ACTION An_Conditions:
//正极纠偏平台允许放料条件
IF  NOT Mach_Control.An_b.An_deviationFalg AND arrAxisCtrl[AxiseNo.AxisName.AndeviationX1].Status.Homed AND NOT arrAxisCtrl[AxiseNo.AxisName.AndeviationX1].Status.Error AND 
	arrAxisCtrl[AxiseNo.AxisName.AndeviationX1].Status.NoMoving AND arrAxisCtrl[AxiseNo.AxisName.AndeviationX1].Cmd.arrbRealPoint[1] AND 
	arrAxisCtrl[AxiseNo.AxisName.AndeviationX2].Status.Homed AND NOT arrAxisCtrl[AxiseNo.AxisName.AndeviationX2].Status.Error AND 
	arrAxisCtrl[AxiseNo.AxisName.AndeviationX2].Status.NoMoving AND arrAxisCtrl[AxiseNo.AxisName.AndeviationX2].Cmd.arrbRealPoint[1] AND 
	arrAxisCtrl[AxiseNo.AxisName.AndeviationY].Status.Homed AND NOT arrAxisCtrl[AxiseNo.AxisName.AndeviationY].Status.Error AND 
	arrAxisCtrl[AxiseNo.AxisName.AndeviationY].Status.NoMoving AND arrAxisCtrl[AxiseNo.AxisName.AndeviationY].Cmd.arrbRealPoint[1] THEN
	Mach_Control.An_b.An_deviationFPOK:=TRUE;
ELSE
	Mach_Control.An_b.An_deviationFPOK:=FALSE;
END_IF 
(*
//正极纠偏平台允许取料条件
IF Mach_Control.An_b.An_deviationFalg AND  (Mach_Control.An_b.An_deviationDone OR Mach_Control.U.CCD_ChosesHMI OR Mach_Control.U.EmptyRunMode) THEN
	Mach_Control.An_b.An_deviationDPOK:=TRUE;
ELSE
	Mach_Control.An_b.An_deviationDPOK:=FALSE;
END_IF
*)
//正极送片搬运平移在安全位，正极送片升降在安全位，允许正极叠片搬运平移到纠偏位
IF arrAxisCtrl[AxiseNo.AxisName.AnCarryingLine].Status.Homed AND arrAxisCtrl[AxiseNo.AxisName.AnCarryingLine].Status.NoMoving AND arrAxisCtrl[AxiseNo.AxisName.AnCarryingLine].Cmd.arrbRealPoint[1] AND 
 	arrAxisCtrl[AxiseNo.AxisName.AnDTCarryingUpDown].Status.Homed AND arrAxisCtrl[AxiseNo.AxisName.AnDTCarryingUpDown].Status.NoMoving AND arrAxisCtrl[AxiseNo.AxisName.AnDTCarryingUpDown].Cmd.arrbRealPoint[1] THEN
	Mach_Control.An_b.CarryingSafepos[0]:=TRUE;
ELSE
	Mach_Control.An_b.CarryingSafepos[0]:=FALSE;
END_IF
//正极隔膜平移在负极片位、正极送片搬运升降在安全位，允许正极叠片搬动至叠台位
IF arrAxisCtrl[AxiseNo.AxisName.SEPTATLine].Status.Homed AND arrAxisCtrl[AxiseNo.AxisName.SEPTATLine].Status.NoMoving AND arrAxisCtrl[AxiseNo.AxisName.SEPTATLine].Cmd.arrbRealPoint[2] AND 
	 	arrAxisCtrl[AxiseNo.AxisName.AnDTCarryingUpDown].Status.Homed AND arrAxisCtrl[AxiseNo.AxisName.AnDTCarryingUpDown].Status.NoMoving AND arrAxisCtrl[AxiseNo.AxisName.AnDTCarryingUpDown].Cmd.arrbRealPoint[1] THEN
	Mach_Control.An_b.CarryingSafepos[1]:=TRUE;
ELSE		
	Mach_Control.An_b.CarryingSafepos[1]:=FALSE;
END_IF
//正极送片搬运升降在安全位，允许正极送片搬运平移至取流水线极片位
IF  arrAxisCtrl[AxiseNo.AxisName.AnCarryingUpDown].Status.Homed AND arrAxisCtrl[AxiseNo.AxisName.AnCarryingUpDown].Status.NoMoving AND arrAxisCtrl[AxiseNo.AxisName.AnCarryingUpDown].Cmd.arrbRealPoint[1] THEN
		Mach_Control.An_b.CarryingSafepos[2]:=TRUE;
ELSE
		Mach_Control.An_b.CarryingSafepos[2]:=FALSE;	
END_IF
//正极送片搬运升降在安全位、正极叠片搬运平移在安全位，允许正极送片搬运平移纠偏位
IF  arrAxisCtrl[AxiseNo.AxisName.AnCarryingUpDown].Status.Homed AND arrAxisCtrl[AxiseNo.AxisName.AnCarryingUpDown].Status.NoMoving AND arrAxisCtrl[AxiseNo.AxisName.AnCarryingUpDown].Cmd.arrbRealPoint[1] AND 
 	arrAxisCtrl[AxiseNo.AxisName.AnDTCarryingLine].Status.Homed AND arrAxisCtrl[AxiseNo.AxisName.AnDTCarryingLine].Status.NoMoving AND arrAxisCtrl[AxiseNo.AxisName.AnDTCarryingLine].Cmd.arrbRealPoint[2]  THEN
		Mach_Control.An_b.CarryingSafepos[3]:=TRUE;
ELSE
		Mach_Control.An_b.CarryingSafepos[3]:=FALSE;	
END_IF
//允许正极纠偏平台移动
IF arrAxisCtrl[AxiseNo.AxisName.AnCarryingUpDown].Status.Homed AND arrAxisCtrl[AxiseNo.AxisName.AnCarryingLine].Status.Homed AND 
	((arrAxisCtrl[AxiseNo.AxisName.AnCarryingUpDown].Status.fSetPos<=arrAxisPar[AxiseNo.AxisName.AnCarryingUpDown].arrTargetPoint[4]+2) OR arrAxisCtrl[AxiseNo.AxisName.AnCarryingLine].Cmd.arrbGoSetPos[1]) AND 
	((arrAxisCtrl[AxiseNo.AxisName.AnDTCarryingUpDown].Status.fSetPos<=arrAxisPar[AxiseNo.AxisName.AnDTCarryingUpDown].arrTargetPoint[4]+2) OR arrAxisCtrl[AxiseNo.AxisName.AnDTCarryingLine].Cmd.arrbGoSetPos[2])THEN
	Mach_Control.An_b.CarryingSafepos[4]:=TRUE;
ELSE
	Mach_Control.An_b.CarryingSafepos[4]:=FALSE;
END_IF
//正极取流水线机械手在安全位，允许模切流水线移动
(*
IF arrAxisCtrl[AxiseNo.AxisName.AnCarryingUpDown].Status.Homed AND NOT Mach_Control.An_b.An_MainBelting AND
	(arrAxisCtrl[AxiseNo.AxisName.AnCarryingUpDown].Status.fSetPos<=arrAxisPar[AxiseNo.AxisName.AnCarryingUpDown].arrTargetPoint[4]+0.2 OR arrAxisCtrl[AxiseNo.AxisName.AnCarryingLine].Cmd.arrbRealPoint[2]) THEN
	Mach_Control.An_b.AN_BeltSafe:=TRUE;
ELSE
	Mach_Control.An_b.AN_BeltSafe:=FALSE;
END_IF
*)
(*
IF  Mach_Control.An_b.An_MainBelting  THEN
	Mach_Control.An_b.AN_BeltSafe:=TRUE;
ELSIF NOT Mach_Control.An_b.An_MainBelting AND  arrAxisCtrl[AxiseNo.AxisName.AnCarryingUpDown].Cmd.arrbRealPoint[4] THEN
	Mach_Control.An_b.AN_BeltSafe:=FALSE;
END_IF
*)
IF  Mach_Control.An_b.An_MainBelting  THEN
	Mach_Control.An_b.AN_BeltSafe:=TRUE;
ELSE
	Mach_Control.An_b.AN_BeltSafe:=FALSE;
END_IF

//正极主流水线取片完成延时复位
An_BeltTon(IN:=Mach_Control.An_b.AN_BeltDone , PT:=T#0.1S , Q=> , ET=> );
IF An_BeltTon.Q THEN
	Mach_Control.An_b.AN_BeltDone :=FALSE;
END_IF


//正极跳取条件1:空跑(空叠隔膜)
An_JumpRules[1]:=Mach_Control.U.EmptyRunMode OR (Mach_Control.DT_b.SinStepMode AND An_Step0<>150);
//正极跳取条件2:手动
An_JumpRules[2]:=Mach_Control.U.DT_iMode<>1;
//正极跳取条件3:叠完电芯后空叠隔膜
An_JumpRules[3]:=Mach_Control.DT_b.DP_Mode AND Mach_Control.An_b.An_Quantited=Par.stDT_date.An_Quantity AND Par.stDT_date.An_Quantity<>0  ;
//正极跳取条件4:叠完电芯后下料
An_JumpRules[4]:=DP_Step0>=6000;//(DP_Step0>=6030 AND DP_Step0<6041) ;
//正极跳取条件5:正极剔废,
An_JumpRules[5]:=(An_Step2<>0 AND An_Step2<>6666) ; 
//正极跳取条件6:接带、蓝胶判断
An_JumpRules[6]:=Bnt_Blueflaging AND Mach_Control.Ca_b.Ca_Quantited>=Par.stDT_date.DT_Overhang_SUM AND Par.stDT_date.DT_Overhang_SUM>0 
				AND Mach_Control.Ca_b.Ca_Quantited>Mach_Control.An_b.An_Quantited AND An_StandbyStep1<1000;//已经进入取片流程则取完当前片
//正极跳取条件7:取片升降有片
An_JumpRules[7]:= Mach_Control.An_b.An_CarryingFalg  ;
//正极跳取条件8:对齐度踢废
An_JumpRules[8]:=Mach_Control.DT_b.DT_Oerhang_Z=2 AND  Par.stDT_date.DT_Overhang_SUM>0 AND Mach_Control.Ca_b.Ca_Quantited>=Par.stDT_date.DT_Overhang_SUM
				AND Mach_Control.An_b.An_Quantited<Mach_Control.Ca_b.Ca_Quantited  AND  Mach_Control.DT_b.DT_CellNG_TF AND Mach_Control.DT_b.Overhang_TF 
				AND((NOT Mach_Control.DT_b.FirstEmpFold AND   bFirstFoldFinish[1]) OR (Mach_Control.DT_b.FirstEmpFold)) AND An_StandbyStep1<1000;//已经进入取片流程则取完当前片
//正极跳取条件9:负极剔废
An_JumpRules[9]:=(Ca_Step2<>0 AND Ca_Step2<>6666) ;
//正极跳取条件10:首层空叠隔膜流程
An_JumpRules[10]:=NOT bFirstFoldFinish[1]AND NOT Mach_Control.DT_b.FirstEmpFold ; 			
//正极跳取条件
Mach_Control.An_b.JumpPiceReady:=An_JumpRules[1] OR An_JumpRules[2] OR An_JumpRules[3] OR An_JumpRules[4] OR An_JumpRules[5]
				OR An_JumpRules[6] OR An_JumpRules[7] OR An_JumpRules[8]  OR An_JumpRules[9] OR An_JumpRules[10] OR DP_Step0=162;	//速度不一样如果平移没到位放弃取片 20240509 CF	
//正极取片条件
Mach_Control.An_b.GetPiceReady:=NOT Mach_Control.An_b.JumpPiceReady (*AND  arrAxisCtrl[AxiseNo.AxisName.AnCarryingUpDown].Cmd.arrbRealPoint[4]*)
				AND ABS(arrAxisCtrl[AxiseNo.AxisName.AnCarryingLine].Status.fSetPos-arrAxisPar[AxiseNo.AxisName.AnCarryingLine].arrTargetPoint[1])<0.5 AND  arrAxisCtrl[AxiseNo.AxisName.AnCarryingWhirling].Cmd.arrbRealPoint[1]
				AND Mach_Control.U.DT_iMode=1 AND NOT Mach_Control.An_b.An_CarryingFalg ;//20240509 CF 升降位置判断屏蔽
		
(*				
////////////////判断叠台是否需要极片
//南昌原版
JumpPiceReady_temp1:=Mach_Control.An_b.An_Quantited<Mach_Control.Ca_b.Ca_Quantited AND Par.stDT_date.An_Quantity<>0  AND
 	 				 Par.stDT_date.Ca_Quantity <>0 AND  Mach_Control.DT_b.DT_CellNG_TF AND
	 				 Mach_Control.Ca_b.Ca_Quantited>=Par.stDT_date.DT_Overhang_SUM AND Par.stDT_date.DT_Overhang_SUM>0  AND
     				 Mach_Control.DT_b.DT_Oerhang_Z=2 AND  NOT Mach_Control.U.EmptyRunMode;

JumpPiceReady_temp2:=Bnt_Blueflaging AND ((Mach_Control.An_b.An_Quantited=0 AND Mach_Control.Ca_b.Ca_Quantited=0) OR
 					 Mach_Control.Ca_b.Ca_Quantited>Mach_Control.An_b.An_Quantited);

JumpPiceReady_temp3:= Mach_Control.An_b.An_Quantited >= Par.stDT_date.An_Quantity  AND
  					  Mach_Control.Ca_b.Ca_Quantited >= Par.stDT_date.Ca_Quantity AND
                      Par.stDT_date.An_Quantity<>0  AND Par.stDT_date.Ca_Quantity <>0;
					  
JumpPiceReady_temp4:= (Ca_Step2<>0 AND Ca_Step2<>6666 AND Mach_Control.U.DT_iMode=1)OR (Mach_Control.An_b.An_Quantited >= Par.stDT_date.An_Quantity 
					 AND  Mach_Control.Ca_b.Ca_Quantited >= (Par.stDT_date.Ca_Quantity-1)) OR
					   (Bnt_Blueflaging AND Mach_Control.Ca_b.Ca_Quantited>=Par.stDT_date.DT_Overhang_SUM AND Par.stDT_date.DT_Overhang_SUM>0);

					   
//正极送片搬运搬运取片准备好
IF Mach_Control.U.DT_iMode=1 AND NOT Mach_Control.An_b.An_CarryingFalg AND NOT JumpPiceReady_temp4 AND (DP_Step0<>6030 AND DP_Step0<>6040 AND 
Mach_Control.An_b.An_Quantited <= Par.stDT_date.An_Quantity  AND  Mach_Control.Ca_b.Ca_Quantited < Par.stDT_date.Ca_Quantity) AND
   arrAxisCtrl[AxiseNo.AxisName.AnCarryingUpDown].Cmd.arrbRealPoint[4] AND arrAxisCtrl[AxiseNo.AxisName.AnCarryingUpDown].Status.Homed AND
   arrAxisCtrl[AxiseNo.AxisName.AnCarryingLine].Cmd.arrbRealPoint[1] AND arrAxisCtrl[AxiseNo.AxisName.AnCarryingLine].Status.Homed AND
   arrAxisCtrl[AxiseNo.AxisName.AnCarryingWhirling].Cmd.arrbRealPoint[1]AND arrAxisCtrl[AxiseNo.AxisName.AnCarryingWhirling].Status.Homed  THEN
   Mach_Control.An_b.GetPiceReady:=TRUE;
ELSE
   Mach_Control.An_b.GetPiceReady:=FALSE;	
END_IF

//正极送片搬运不取片
IF Mach_Control.U.DT_iMode<>1 OR Mach_Control.An_b.An_CarryingFalg OR JumpPiceReady_temp1 OR JumpPiceReady_temp2 OR JumpPiceReady_temp3 OR JumpPiceReady_temp4 OR Mach_Control.U.EmptyRunMode THEN
	Mach_Control.An_b.JumpPiceReady:=TRUE;
ELSE
	Mach_Control.An_b.JumpPiceReady:=FALSE;	
END_IF


//合肥原版
(*
(********************正极取片准备好********************)															
Mach_Control.An_b.GetPiceReady:=NOT Mach_Control.An_b.JumpPiceReady AND 
							arrAxisCtrl[AxiseNo.AxisName.AnCarryingUpDown].Cmd.arrbRealPoint[4] AND arrAxisCtrl[AxiseNo.AxisName.AnCarryingUpDown].Status.Homed AND
							arrAxisCtrl[AxiseNo.AxisName.AnCarryingLine].Cmd.arrbRealPoint[1] AND arrAxisCtrl[AxiseNo.AxisName.AnCarryingLine].Status.Homed AND
							arrAxisCtrl[AxiseNo.AxisName.AnCarryingWhirling].Cmd.arrbRealPoint[1]AND arrAxisCtrl[AxiseNo.AxisName.AnCarryingWhirling].Status.Homed AND 
							(DP_Step0<>6030 AND DP_Step0<>6040)  ;													

(********************正极放弃取片********************)
Mach_Control.An_b.JumpPiceReady:=Mach_Control.U.DT_iMode<>1 OR Mach_Control.An_b.An_CarryingFalg OR Blueflaging OR Mach_Control.U.EmptyRunMode
															OR Mach_Control.An_b.An_Quantited=Par.stDT_date.An_Quantity;
*)

*)


/////////////////////////////////////////////////////////////
/////////////////////////////////////////////////////////
////////////////////////////////////////////电机条件
//正极送片搬运平移
IF arrAxisCtrl[AxiseNo.AxisName.AnCarryingUpDown].Status.fSetPos<=arrAxisPar[AxiseNo.AxisName.AnCarryingUpDown].arrTargetPoint[4]+1 AND
 	arrAxisCtrl[AxiseNo.AxisName.AnCarryingUpDown].Status.Homed AND arrAxisCtrl[AxiseNo.AxisName.AnCarryingUpDown].Status.NoMoving	AND Mach_Control.U.DT_iMode=3 THEN
arrAxisCtrl[AxiseNo.AxisName.AnCarryingLine].Cmd.Home_Condition:=TRUE;
ELSE
arrAxisCtrl[AxiseNo.AxisName.AnCarryingLine].Cmd.Home_Condition:=FALSE;	
END_IF

IF arrAxisCtrl[AxiseNo.AxisName.AnCarryingUpDown].Status.fSetPos<=arrAxisPar[AxiseNo.AxisName.AnCarryingUpDown].arrTargetPoint[4]+1 AND
	arrAxisCtrl[AxiseNo.AxisName.AnCarryingUpDown].Status.Homed AND arrAxisCtrl[AxiseNo.AxisName.AnCarryingUpDown].Status.NoMoving AND Mach_Control.U.DT_iMode=3 
    AND 	arrCyCtrl[arrCyNo.CylinderName.AnScrapbinCy].Io.DIOnSwitch  THEN
arrAxisCtrl[AxiseNo.AxisName.AnCarryingLine].Cmd.GoPoint_Condition[1]:=TRUE;
ELSE
arrAxisCtrl[AxiseNo.AxisName.AnCarryingLine].Cmd.GoPoint_Condition[1]:=FALSE;	
END_IF

IF arrAxisCtrl[AxiseNo.AxisName.AnCarryingUpDown].Status.fSetPos<=arrAxisPar[AxiseNo.AxisName.AnCarryingUpDown].arrTargetPoint[4]+1 AND arrAxisCtrl[AxiseNo.AxisName.AnCarryingUpDown].Status.Homed  AND
	 arrAxisCtrl[AxiseNo.AxisName.AnCarryingLine].Status.Homed AND Mach_Control.U.DT_iMode=3 AND 	arrCyCtrl[arrCyNo.CylinderName.AnScrapbinCy].Io.DIOnSwitch AND
	 arrAxisCtrl[AxiseNo.AxisName.AnDTCarryingLine].Status.Homed AND arrAxisCtrl[AxiseNo.AxisName.AnDTCarryingLine].Cmd.arrbRealPoint[2] THEN//比较值要根据实际值修改
	arrAxisCtrl[AxiseNo.AxisName.AnCarryingLine].Cmd.GoPoint_Condition[2]:=TRUE;
ELSE
	arrAxisCtrl[AxiseNo.AxisName.AnCarryingLine].Cmd.GoPoint_Condition[2]:=FALSE;	
END_IF

//正极送片搬运升降
IF Mach_Control.U.DT_iMode=3  THEN
	arrAxisCtrl[AxiseNo.AxisName.AnCarryingUpDown].Cmd.Home_Condition:=TRUE;
ELSE
	arrAxisCtrl[AxiseNo.AxisName.AnCarryingUpDown].Cmd.Home_Condition:=FALSE;	
END_IF

IF Mach_Control.U.DT_iMode=3 AND arrAxisCtrl[AxiseNo.AxisName.AnCarryingUpDown].Status.Homed THEN
	arrAxisCtrl[AxiseNo.AxisName.AnCarryingUpDown].Cmd.GoPoint_Condition[1]:=TRUE;
ELSE
	arrAxisCtrl[AxiseNo.AxisName.AnCarryingUpDown].Cmd.GoPoint_Condition[1]:=FALSE;	
END_IF

IF (*arrAxisCtrl[AxiseNo.AxisName.AnCarryingLine].Cmd.arrbRealPoint[1] AND*)  Mach_Control.U.DT_iMode=3 AND arrAxisCtrl[AxiseNo.AxisName.AnCarryingUpDown].Status.Homed THEN
	arrAxisCtrl[AxiseNo.AxisName.AnCarryingUpDown].Cmd.GoPoint_Condition[2]:=TRUE;
ELSE
	arrAxisCtrl[AxiseNo.AxisName.AnCarryingUpDown].Cmd.GoPoint_Condition[2]:=FALSE;	
END_IF

IF (*arrAxisCtrl[AxiseNo.AxisName.AnCarryingLine].Cmd.arrbRealPoint[2] AND*)  Mach_Control.U.DT_iMode=3 AND arrAxisCtrl[AxiseNo.AxisName.AnCarryingUpDown].Status.Homed THEN
	arrAxisCtrl[AxiseNo.AxisName.AnCarryingUpDown].Cmd.GoPoint_Condition[3]:=TRUE;
ELSE
	arrAxisCtrl[AxiseNo.AxisName.AnCarryingUpDown].Cmd.GoPoint_Condition[3]:=FALSE;	
END_IF

IF (*arrAxisCtrl[AxiseNo.AxisName.AnCarryingLine].Cmd.arrbRealPoint[1] AND*)  Mach_Control.U.DT_iMode=3 AND arrAxisCtrl[AxiseNo.AxisName.AnCarryingUpDown].Status.Homed THEN
	arrAxisCtrl[AxiseNo.AxisName.AnCarryingUpDown].Cmd.GoPoint_Condition[4]:=TRUE;
ELSE
	arrAxisCtrl[AxiseNo.AxisName.AnCarryingUpDown].Cmd.GoPoint_Condition[4]:=FALSE;	
END_IF

//正极送片搬运旋转
IF Mach_Control.U.DT_iMode=3 AND
 	arrAxisCtrl[AxiseNo.AxisName.AnCarryingUpDown].Status.fSetPos <= arrAxisPar[AxiseNo.AxisName.AnCarryingUpDown].arrTargetPoint[1]+1 AND 
	arrAxisCtrl[AxiseNo.AxisName.AnCarryingUpDown].Status.Homed AND arrCyCtrl[arrCyNo.CylinderName.AnScrapbinCy].Io.DIOnSwitch   THEN
	arrAxisCtrl[AxiseNo.AxisName.AnCarryingWhirling].Cmd.Home_Condition:=TRUE;
ELSE
	arrAxisCtrl[AxiseNo.AxisName.AnCarryingWhirling].Cmd.Home_Condition:=FALSE;	
END_IF


IF Mach_Control.U.DT_iMode=3 AND
 	arrAxisCtrl[AxiseNo.AxisName.AnCarryingUpDown].Status.fSetPos <= arrAxisPar[AxiseNo.AxisName.AnCarryingUpDown].arrTargetPoint[1]+1 AND 
	arrAxisCtrl[AxiseNo.AxisName.AnCarryingUpDown].Status.Homed AND arrCyCtrl[arrCyNo.CylinderName.AnScrapbinCy].Io.DIOnSwitch    THEN
	   arrAxisCtrl[AxiseNo.AxisName.AnCarryingWhirling].Cmd.JogP_Condition:=TRUE;
	   arrAxisCtrl[AxiseNo.AxisName.AnCarryingWhirling].Cmd.JogN_Condition:=TRUE;
 ELSE 
	   arrAxisCtrl[AxiseNo.AxisName.AnCarryingWhirling].Cmd.JogP_Condition:=FALSE;
	   arrAxisCtrl[AxiseNo.AxisName.AnCarryingWhirling].Cmd.JogN_Condition:=FALSE;
 END_IF

IF Mach_Control.U.DT_iMode=3 AND 
	(arrAxisCtrl[AxiseNo.AxisName.AnCarryingUpDown].Cmd.arrbRealPoint[1] (*OR arrAxisCtrl[AxiseNo.AxisName.AnCarryingUpDown].Cmd.arrbRealPoint[4]*))AND
	arrAxisCtrl[AxiseNo.AxisName.AnCarryingUpDown].Status.Homed AND arrAxisCtrl[AxiseNo.AxisName.AnCarryingWhirling].Status.Homed AND 
    arrCyCtrl[arrCyNo.CylinderName.AnScrapbinCy].Io.DIOnSwitch   THEN
	arrAxisCtrl[AxiseNo.AxisName.AnCarryingWhirling].Cmd.GoPoint_Condition[1]:=TRUE;
ELSE
	arrAxisCtrl[AxiseNo.AxisName.AnCarryingWhirling].Cmd.GoPoint_Condition[1]:=FALSE;	
END_IF

IF Mach_Control.U.DT_iMode=3 AND 
	(arrAxisCtrl[AxiseNo.AxisName.AnCarryingUpDown].Cmd.arrbRealPoint[1] (*OR arrAxisCtrl[AxiseNo.AxisName.AnCarryingUpDown].Cmd.arrbRealPoint[4]*)) AND
	arrAxisCtrl[AxiseNo.AxisName.AnCarryingUpDown].Status.Homed AND arrAxisCtrl[AxiseNo.AxisName.AnCarryingWhirling].Status.Homed AND
   arrCyCtrl[arrCyNo.CylinderName.AnScrapbinCy].Io.DIOnSwitch  THEN
	arrAxisCtrl[AxiseNo.AxisName.AnCarryingWhirling].Cmd.GoPoint_Condition[2]:=TRUE;
ELSE
	arrAxisCtrl[AxiseNo.AxisName.AnCarryingWhirling].Cmd.GoPoint_Condition[2]:=FALSE;	
END_IF

//正极纠偏平台X1
IF Mach_Control.U.DT_iMode=3  OR  (DP_Step0>=6015 AND   DP_Step0<=6041)   THEN
	arrAxisCtrl[AxiseNo.AxisName.AndeviationX1].Cmd.Home_Condition:=TRUE;
ELSE
	arrAxisCtrl[AxiseNo.AxisName.AndeviationX1].Cmd.Home_Condition:=FALSE;	
END_IF

IF Mach_Control.U.DT_iMode=3 AND arrAxisCtrl[AxiseNo.AxisName.AndeviationX1].Status.Homed THEN
	arrAxisCtrl[AxiseNo.AxisName.AndeviationX1].Cmd.GoPoint_Condition[1]:=TRUE;
ELSE
	arrAxisCtrl[AxiseNo.AxisName.AndeviationX1].Cmd.GoPoint_Condition[1]:=FALSE;	
END_IF

IF Mach_Control.U.DT_iMode=3 AND arrAxisCtrl[AxiseNo.AxisName.AndeviationX1].Status.Homed THEN
	arrAxisCtrl[AxiseNo.AxisName.AndeviationX1].Cmd.GoPoint_Condition[2]:=TRUE;
ELSE
	arrAxisCtrl[AxiseNo.AxisName.AndeviationX1].Cmd.GoPoint_Condition[2]:=FALSE;	
END_IF

IF Mach_Control.U.DT_iMode=3 AND arrAxisCtrl[AxiseNo.AxisName.AndeviationX1].Status.Homed THEN
	arrAxisCtrl[AxiseNo.AxisName.AndeviationX1].Cmd.GoPoint_Condition[3]:=TRUE;
ELSE
	arrAxisCtrl[AxiseNo.AxisName.AndeviationX1].Cmd.GoPoint_Condition[3]:=FALSE;	
END_IF

IF Mach_Control.U.DT_iMode=3 AND arrAxisCtrl[AxiseNo.AxisName.AndeviationX1].Status.Homed THEN
	arrAxisCtrl[AxiseNo.AxisName.AndeviationX1].Cmd.GoPoint_Condition[4]:=TRUE;
ELSE
	arrAxisCtrl[AxiseNo.AxisName.AndeviationX1].Cmd.GoPoint_Condition[4]:=FALSE;	
END_IF

IF Mach_Control.U.DT_iMode=3 AND arrAxisCtrl[AxiseNo.AxisName.AndeviationX1].Status.Homed THEN
	arrAxisCtrl[AxiseNo.AxisName.AndeviationX1].Cmd.GoPoint_Condition[5]:=TRUE;
ELSE
	arrAxisCtrl[AxiseNo.AxisName.AndeviationX1].Cmd.GoPoint_Condition[5]:=FALSE;	
END_IF

//正极纠偏平台X2
IF Mach_Control.U.DT_iMode=3  OR  (DP_Step0>=6015 AND   DP_Step0<=6041)   THEN
	arrAxisCtrl[AxiseNo.AxisName.AndeviationX2].Cmd.Home_Condition:=TRUE;
ELSE
	arrAxisCtrl[AxiseNo.AxisName.AndeviationX2].Cmd.Home_Condition:=FALSE;	
END_IF

IF Mach_Control.U.DT_iMode=3 AND arrAxisCtrl[AxiseNo.AxisName.AndeviationX2].Status.Homed THEN
	arrAxisCtrl[AxiseNo.AxisName.AndeviationX2].Cmd.GoPoint_Condition[1]:=TRUE;
ELSE
	arrAxisCtrl[AxiseNo.AxisName.AndeviationX2].Cmd.GoPoint_Condition[1]:=FALSE;	
END_IF

IF Mach_Control.U.DT_iMode=3 AND arrAxisCtrl[AxiseNo.AxisName.AndeviationX2].Status.Homed THEN
	arrAxisCtrl[AxiseNo.AxisName.AndeviationX2].Cmd.GoPoint_Condition[2]:=TRUE;
ELSE
	arrAxisCtrl[AxiseNo.AxisName.AndeviationX2].Cmd.GoPoint_Condition[2]:=FALSE;	
END_IF

IF Mach_Control.U.DT_iMode=3 AND arrAxisCtrl[AxiseNo.AxisName.AndeviationX2].Status.Homed THEN
	arrAxisCtrl[AxiseNo.AxisName.AndeviationX2].Cmd.GoPoint_Condition[3]:=TRUE;
ELSE
	arrAxisCtrl[AxiseNo.AxisName.AndeviationX2].Cmd.GoPoint_Condition[3]:=FALSE;	
END_IF

IF Mach_Control.U.DT_iMode=3 AND arrAxisCtrl[AxiseNo.AxisName.AndeviationX2].Status.Homed THEN
	arrAxisCtrl[AxiseNo.AxisName.AndeviationX2].Cmd.GoPoint_Condition[4]:=TRUE;
ELSE
	arrAxisCtrl[AxiseNo.AxisName.AndeviationX2].Cmd.GoPoint_Condition[4]:=FALSE;	
END_IF

IF Mach_Control.U.DT_iMode=3 AND arrAxisCtrl[AxiseNo.AxisName.AndeviationX2].Status.Homed THEN
	arrAxisCtrl[AxiseNo.AxisName.AndeviationX2].Cmd.GoPoint_Condition[5]:=TRUE;
ELSE
	arrAxisCtrl[AxiseNo.AxisName.AndeviationX2].Cmd.GoPoint_Condition[5]:=FALSE;	
END_IF

//正极纠偏平台Y
IF Mach_Control.U.DT_iMode=3  OR  (DP_Step0>=6015 AND   DP_Step0<=6041)   THEN
	arrAxisCtrl[AxiseNo.AxisName.AndeviationY].Cmd.Home_Condition:=TRUE;
ELSE
	arrAxisCtrl[AxiseNo.AxisName.AndeviationY].Cmd.Home_Condition:=FALSE;	
END_IF

IF Mach_Control.U.DT_iMode=3 AND arrAxisCtrl[AxiseNo.AxisName.AndeviationY].Status.Homed THEN
	arrAxisCtrl[AxiseNo.AxisName.AndeviationY].Cmd.GoPoint_Condition[1]:=TRUE;
ELSE
	arrAxisCtrl[AxiseNo.AxisName.AndeviationY].Cmd.GoPoint_Condition[1]:=FALSE;	
END_IF

IF Mach_Control.U.DT_iMode=3 AND arrAxisCtrl[AxiseNo.AxisName.AndeviationY].Status.Homed THEN
	arrAxisCtrl[AxiseNo.AxisName.AndeviationY].Cmd.GoPoint_Condition[2]:=TRUE;
ELSE
	arrAxisCtrl[AxiseNo.AxisName.AndeviationY].Cmd.GoPoint_Condition[2]:=FALSE;	
END_IF

IF Mach_Control.U.DT_iMode=3 AND arrAxisCtrl[AxiseNo.AxisName.AndeviationY].Status.Homed THEN
	arrAxisCtrl[AxiseNo.AxisName.AndeviationY].Cmd.GoPoint_Condition[3]:=TRUE;
ELSE
	arrAxisCtrl[AxiseNo.AxisName.AndeviationY].Cmd.GoPoint_Condition[3]:=FALSE;	
END_IF

IF Mach_Control.U.DT_iMode=3 AND arrAxisCtrl[AxiseNo.AxisName.AndeviationY].Status.Homed THEN
	arrAxisCtrl[AxiseNo.AxisName.AndeviationY].Cmd.GoPoint_Condition[4]:=TRUE;
ELSE
	arrAxisCtrl[AxiseNo.AxisName.AndeviationY].Cmd.GoPoint_Condition[4]:=FALSE;	
END_IF

IF Mach_Control.U.DT_iMode=3 AND arrAxisCtrl[AxiseNo.AxisName.AndeviationY].Status.Homed THEN
	arrAxisCtrl[AxiseNo.AxisName.AndeviationY].Cmd.GoPoint_Condition[5]:=TRUE;
ELSE
	arrAxisCtrl[AxiseNo.AxisName.AndeviationY].Cmd.GoPoint_Condition[5]:=FALSE;	
END_IF

//正极叠台搬运平移1
IF Mach_Control.U.DT_iMode=3 AND arrAxisCtrl[AxiseNo.AxisName.AnDTCarryingUpDown].Status.Homed AND
	arrAxisCtrl[AxiseNo.AxisName.AnDTCarryingUpDown].Status.fSetPos<= arrAxisPar[AxiseNo.AxisName.AnDTCarryingUpDown].arrTargetPoint[4]+1 AND
	arrAxisCtrl[AxiseNo.AxisName.AnCarryingLine].Status.fSetPos<=arrAxisPar[AxiseNo.AxisName.AnCarryingLine].arrTargetPoint[1] AND 
	arrCyCtrl[arrCyNo.CylinderName.AnScrapbinCy].Io.DIOnSwitch  AND NOT arrCyCtrl[arrCyNo.CylinderName.AnScrapbinCy].Io.DIOFFSwitch AND
	arrAxisCtrl[AxiseNo.AxisName.AnCarryingLine].Status.Homed AND arrAxisCtrl[AxiseNo.AxisName.AnCarryingLine].Status.NoMoving THEN
	arrAxisCtrl[AxiseNo.AxisName.AnDTCarryingLine].Cmd.Home_Condition:=TRUE;
ELSE
	arrAxisCtrl[AxiseNo.AxisName.AnDTCarryingLine].Cmd.Home_Condition:=FALSE;	
END_IF

IF Mach_Control.U.DT_iMode=3 AND arrCyCtrl[arrCyNo.CylinderName.AnScrapbinCy].Status.ONState THEN
   arrAxisCtrl[AxiseNo.AxisName.AnDTCarryingLine].Cmd.JogP_Condition:=TRUE;
   arrAxisCtrl[AxiseNo.AxisName.AnDTCarryingLine].Cmd.JogN_Condition:=TRUE;
   ELSE 
   arrAxisCtrl[AxiseNo.AxisName.AnDTCarryingLine].Cmd.JogP_Condition:=FALSE;
   arrAxisCtrl[AxiseNo.AxisName.AnDTCarryingLine].Cmd.JogN_Condition:=FALSE;
 END_IF

IF Mach_Control.U.DT_iMode=3 AND arrAxisCtrl[AxiseNo.AxisName.AnDTCarryingUpDown].Status.Homed AND
	arrAxisCtrl[AxiseNo.AxisName.AnDTCarryingUpDown].Status.fSetPos<= arrAxisPar[AxiseNo.AxisName.AnDTCarryingUpDown].arrTargetPoint[4]+1 AND
	arrAxisCtrl[AxiseNo.AxisName.AnCarryingLine].Cmd.arrbRealPoint[1] AND arrCyCtrl[arrCyNo.CylinderName.AnScrapbinCy].Status.ONState  THEN
	arrAxisCtrl[AxiseNo.AxisName.AnDTCarryingLine].Cmd.GoPoint_Condition[1]:=TRUE;
ELSE
	arrAxisCtrl[AxiseNo.AxisName.AnDTCarryingLine].Cmd.GoPoint_Condition[1]:=FALSE;	
END_IF

IF Mach_Control.U.DT_iMode=3 AND arrAxisCtrl[AxiseNo.AxisName.AnDTCarryingUpDown].Status.Homed AND
	arrAxisCtrl[AxiseNo.AxisName.AnDTCarryingUpDown].Status.fSetPos<= arrAxisPar[AxiseNo.AxisName.AnDTCarryingUpDown].arrTargetPoint[4]+1 AND
 	arrAxisCtrl[AxiseNo.AxisName.AnDTCarryingLine].Status.Homed AND arrAxisCtrl[AxiseNo.AxisName.SEPTATLine].Cmd.arrbRealPoint[2] AND
    arrCyCtrl[arrCyNo.CylinderName.AnScrapbinCy].Status.ONState THEN
	arrAxisCtrl[AxiseNo.AxisName.AnDTCarryingLine].Cmd.GoPoint_Condition[2]:=TRUE;
ELSE
	arrAxisCtrl[AxiseNo.AxisName.AnDTCarryingLine].Cmd.GoPoint_Condition[2]:=FALSE;	
END_IF


//正极叠台搬运升降1
IF Mach_Control.U.DT_iMode=3  THEN
	arrAxisCtrl[AxiseNo.AxisName.AnDTCarryingUpDown].Cmd.Home_Condition:=TRUE;
ELSE
	arrAxisCtrl[AxiseNo.AxisName.AnDTCarryingUpDown].Cmd.Home_Condition:=FALSE;	
END_IF

IF Mach_Control.U.DT_iMode=3 AND arrAxisCtrl[AxiseNo.AxisName.AnDTCarryingUpDown].Status.Homed THEN
	arrAxisCtrl[AxiseNo.AxisName.AnDTCarryingUpDown].Cmd.GoPoint_Condition[1]:=TRUE;
ELSE
	arrAxisCtrl[AxiseNo.AxisName.AnDTCarryingUpDown].Cmd.GoPoint_Condition[1]:=FALSE;	
END_IF

IF Mach_Control.U.DT_iMode=3 AND  arrAxisCtrl[AxiseNo.AxisName.AnDTCarryingUpDown].Status.Homed THEN
	arrAxisCtrl[AxiseNo.AxisName.AnDTCarryingUpDown].Cmd.GoPoint_Condition[2]:=TRUE;
ELSE
	arrAxisCtrl[AxiseNo.AxisName.AnDTCarryingUpDown].Cmd.GoPoint_Condition[2]:=FALSE;	
END_IF

IF Mach_Control.U.DT_iMode=3 AND arrAxisCtrl[AxiseNo.AxisName.AnDTCarryingUpDown].Status.Homed THEN
	arrAxisCtrl[AxiseNo.AxisName.AnDTCarryingUpDown].Cmd.GoPoint_Condition[3]:=TRUE;
ELSE
	arrAxisCtrl[AxiseNo.AxisName.AnDTCarryingUpDown].Cmd.GoPoint_Condition[3]:=FALSE;	
END_IF

IF Mach_Control.U.DT_iMode=3 AND arrAxisCtrl[AxiseNo.AxisName.AnDTCarryingUpDown].Status.Homed THEN
	arrAxisCtrl[AxiseNo.AxisName.AnDTCarryingUpDown].Cmd.GoPoint_Condition[4]:=TRUE;
ELSE
	arrAxisCtrl[AxiseNo.AxisName.AnDTCarryingUpDown].Cmd.GoPoint_Condition[4]:=FALSE;	
END_IF

IF Mach_Control.U.DT_iMode=3 AND arrAxisCtrl[AxiseNo.AxisName.AnDTCarryingUpDown].Status.Homed THEN
	arrAxisCtrl[AxiseNo.AxisName.AnDTCarryingUpDown].Cmd.GoPoint_Condition[5]:=TRUE;
ELSE
	arrAxisCtrl[AxiseNo.AxisName.AnDTCarryingUpDown].Cmd.GoPoint_Condition[5]:=FALSE;	
END_IF
//正极NG料盒伸缩气缸条件
IF arrAxisCtrl[AxiseNo.AxisName.AnDTCarryingUpDown].Cmd.arrbRealPoint[5] (*AND arrAxisCtrl[AxiseNo.AxisName.AnCarryingLine].Cmd.arrbRealPoint[1]*)  THEN
	arrCyCtrl[arrCyNo.CylinderName.	AnScrapbinCy].Cmd.OnCondition:=TRUE;
    arrCyCtrl[arrCyNo.CylinderName.	AnScrapbinCy].Cmd.OffCondition:=TRUE;
ELSE	
	arrCyCtrl[arrCyNo.CylinderName.	AnScrapbinCy].Cmd.OnCondition:=FALSE;
    arrCyCtrl[arrCyNo.CylinderName.	AnScrapbinCy].Cmd.OffCondition:=FALSE;	
END_IF
END_ACTION

ACTION An_Gohome:
An_GohomeTon(IN:= , PT:=T#1S , Q=> , ET=> );//正极取片回原点延时
An_GohomeOverTon(IN:= , PT:=T#90S , Q=> , ET=> );//负正回原点超时报警延时
rAn_Gohome_TRIG(CLK:=Mach_Control.An_b.An_GohomeHMI , Q=> );//正极取片回原点启动
fAn_Gohome_FRIG(CLK:=Mach_Control.An_b.An_GohomeHMI , Q=> );//负极回原点启动
//判断正极是否回原点完成
IF arrAxisCtrl[AxiseNo.AxisName.AnCarryingUpDown].Status.Homed AND  arrAxisCtrl[AxiseNo.AxisName.AnDTCarryingUpDown].Status.Homed  AND 
 	arrAxisCtrl[AxiseNo.AxisName.AnCarryingLine].Status.Homed AND arrAxisCtrl[AxiseNo.AxisName.AnCarryingWhirling].Status.Homed AND 				
	arrAxisCtrl[AxiseNo.AxisName.AndeviationX1].Status.Homed AND arrAxisCtrl[AxiseNo.AxisName.AndeviationX2].Status.Homed AND
	arrAxisCtrl[AxiseNo.AxisName.AndeviationY].Status.Homed	AND arrAxisCtrl[AxiseNo.AxisName.AnDTCarryingLine].Status.Homed AND An_GohomeDone THEN	
		Mach_Control.An_b.An_GohomeDone:=TRUE;//负极取片回原点完成
ELSE
		Mach_Control.An_b.An_GohomeDone:=FALSE;//负极取片回原点完成
END_IF




IF Mach_Control.U.DT_iMode=3 THEN//在手动状态下
		IF rAn_Gohome_TRIG.Q THEN
			Step_InitAnDT:=0;
			An_GohomeDone:=FALSE;
			An_Gohoming:=FALSE;//负极取片回原点中
			Mach_Control.An_b.An_GohomeDone:=FALSE;//负极取片回原点完成
		END_IF	
END_IF		
IF Mach_Control.U.DT_iMode=3 THEN//在手动状态下
	
//回原点超时报警	

IF  An_Gohoming THEN
		IF 	NOT An_GohomeOverTon.Q THEN
			    An_GohomeOverTon.IN:=TRUE;
		ELSE
			IF 	 An_GohomeOverTon.Q THEN
				An_Gohoming:=FALSE;
			     Mach_Control.An_b.Error[19]:=TRUE;//负极回原点超时报警
			     An_GohomeOverTon.IN:=FALSE;
			END_IF	 
				 
		END_IF

ELSE
		An_GohomeOverTon.IN:=FALSE;
END_IF




//正极取料机构初始C化
CASE Step_InitAnDT OF
0://等待正极回原点启动	
IF fAn_Gohome_FRIG.Q THEN
	An_Gohoming:=TRUE;//负极取片回原点中
	Mach_Control.An_b.An_GohomeHMI:=FALSE;
	Step_InitAnDT:=1;
END_IF
1://复位回原点完成
	An_GohomeDone:=FALSE;//正极回原点完成
	An_GohomeTon.IN:=FALSE;								
	IF NOT An_GohomeDone THEN
		Step_InitAnDT:=10;
	END_IF
10:
Mach_Control.An_b.An_CarryingFalg:=FALSE;//正极搬运升降有料标记
Mach_Control.An_b.An_DPCarryingFalg:=FALSE;//正极叠片搬运有料标记
Mach_Control.An_b.An_deviationFalg :=FALSE;//正极纠偏有料标记


An_StandbyStep0:=0;//正极纠偏平台自动步
An_StandbyStep1:=0;//正极取片备料步清零
An_StandbyStep2:=0;//叠正极片，判断真空、破真空
An_StandbyStep3:=0;//叠正极片，判断主轴是否完成
Mach_Control.An_b.AN_BeltDone:=FALSE;//取流水线取极片完成	
Mach_Control.An_b.An_MainBelting:=FALSE;// 复位正极搬运升降取极片中
An_Step0:=0;
An_Step1:=0;
An_Step2:=0;
An_Step3:=0;
An_StandbyStep0:=0;
An_Demarcate_Step0:=0;
An_RecdevPla_Step0:=0;						
Step_InitAnDT:=20;	
20:
	fbAnCamInCarryingLine.bCamInExecute:=FALSE;//正极送片搬运平移
	fbAnCamInCarryingUpDown.bCamInExecute:=FALSE;//正极送片搬运升降
	fbAnCamInCarryingWhirling.bCamInExecute:=FALSE;//正极送片搬运旋转
	fbAnCamInDTCarryingLine.bCamInExecute:=FALSE;//正极叠片搬运平移
	fbAnCamInDTCarryingUpDown.bCamInExecute:=FALSE;//正极叠片搬运升降
	IF NOT fbAnCamInCarryingLine.bCamInExecute AND NOT fbAnCamInCarryingUpDown.bCamInExecute AND 
		NOT  fbAnCamInCarryingWhirling.bCamInExecute AND NOT fbAnCamInDTCarryingLine.bCamInExecute AND 
		NOT  fbAnCamInDTCarryingUpDown.bCamInExecute THEN
				Step_InitAnDT:=25;	
	END_IF									
25:
arrAxisCtrl[AxiseNo.AxisName.AnCarryingUpDown].Cmd.bHalt:=TRUE;//正极送片搬运轴解耦
arrAxisCtrl[AxiseNo.AxisName.AnDTCarryingUpDown].Cmd.bHalt:=TRUE;//正极叠片搬运解耦
arrAxisCtrl[AxiseNo.AxisName.AnCarryingLine].Cmd.bHalt:=TRUE;//正极送片搬运平移轴解耦
arrAxisCtrl[AxiseNo.AxisName.AnDTCarryingLine].Cmd.bHalt:=TRUE;//正极叠片搬运平移轴解耦
arrAxisCtrl[AxiseNo.AxisName.AnCarryingWhirling].Cmd.bHalt:=TRUE;//正极送片搬运旋转轴解耦	
IF NOT arrAxisCtrl[AxiseNo.AxisName.AnCarryingUpDown].Status.Coupled AND arrAxisCtrl[AxiseNo.AxisName.AnCarryingUpDown].Status.NoMoving AND 
   NOT arrAxisCtrl[AxiseNo.AxisName.AnDTCarryingUpDown].Status.Coupled AND arrAxisCtrl[AxiseNo.AxisName.AnDTCarryingUpDown].Status.NoMoving AND
   NOT arrAxisCtrl[AxiseNo.AxisName.AnCarryingLine].Status.Coupled AND arrAxisCtrl[AxiseNo.AxisName.AnCarryingLine].Status.NoMoving AND 
   NOT arrAxisCtrl[AxiseNo.AxisName.AnDTCarryingLine].Status.Coupled AND arrAxisCtrl[AxiseNo.AxisName.AnDTCarryingLine].Status.NoMoving AND
   NOT arrAxisCtrl[AxiseNo.AxisName.AnCarryingWhirling].Status.Coupled AND arrAxisCtrl[AxiseNo.AxisName.AnCarryingWhirling].Status.NoMoving THEN
			arrAxisCtrl[AxiseNo.AxisName.AnCarryingUpDown].Cmd.bHalt:=FALSE;//正极送片搬运轴解耦
			arrAxisCtrl[AxiseNo.AxisName.AnDTCarryingUpDown].Cmd.bHalt:=FALSE;//正极叠片搬运解耦
			arrAxisCtrl[AxiseNo.AxisName.AnCarryingLine].Cmd.bHalt:=FALSE;//正极送片搬运平移轴解耦
			arrAxisCtrl[AxiseNo.AxisName.AnDTCarryingLine].Cmd.bHalt:=FALSE;//正极叠片搬运平移轴解耦
			arrAxisCtrl[AxiseNo.AxisName.AnCarryingWhirling].Cmd.bHalt:=FALSE;//正极送片搬运旋转轴解耦	
			Step_InitAnDT:=30;	
END_IF		
30:
arrAxisCtrl[AxiseNo.AxisName.AnCarryingUpDown].Cmd.bEnable:=TRUE;//正极送片搬运轴
arrAxisCtrl[AxiseNo.AxisName.AnDTCarryingUpDown].Cmd.bEnable:=TRUE;//正极叠片搬运
arrAxisCtrl[AxiseNo.AxisName.AnCarryingLine].Cmd.bEnable:=TRUE;//正极送片搬运平移轴
arrAxisCtrl[AxiseNo.AxisName.AnDTCarryingLine].Cmd.bEnable:=TRUE;//正极叠片搬运平移轴
arrAxisCtrl[AxiseNo.AxisName.AnCarryingWhirling].Cmd.bEnable:=TRUE;//正极送片搬运旋转轴	
arrAxisCtrl[AxiseNo.AxisName.AndeviationX1].Cmd.bEnable:=TRUE;//正极纠偏X1
arrAxisCtrl[AxiseNo.AxisName.AndeviationX2].Cmd.bEnable:=TRUE;//正极纠偏X2
arrAxisCtrl[AxiseNo.AxisName.AndeviationY].Cmd.bEnable:=TRUE;//正极纠偏Y						
IF arrAxisCtrl[AxiseNo.AxisName.AnCarryingUpDown].Status.Enabled AND 
   arrAxisCtrl[AxiseNo.AxisName.AnDTCarryingUpDown].Status.Enabled AND 
   arrAxisCtrl[AxiseNo.AxisName.AnCarryingLine].Status.Enabled AND 
   arrAxisCtrl[AxiseNo.AxisName.AnDTCarryingLine].Status.Enabled AND 
   arrAxisCtrl[AxiseNo.AxisName.AnCarryingWhirling].Status.Enabled AND
   arrAxisCtrl[AxiseNo.AxisName.AndeviationX1].Status.Enabled AND 
   arrAxisCtrl[AxiseNo.AxisName.AndeviationX2].Status.Enabled AND
   arrAxisCtrl[AxiseNo.AxisName.AndeviationY].Status.Enabled THEN
		Step_InitAnDT:=35;	
ELSIF arrAxisCtrl[AxiseNo.AxisName.AnCarryingUpDown].Status.Error OR 
   arrAxisCtrl[AxiseNo.AxisName.AnDTCarryingUpDown].Status.Error OR 
   arrAxisCtrl[AxiseNo.AxisName.AnCarryingLine].Status.Error OR 
   arrAxisCtrl[AxiseNo.AxisName.AnDTCarryingLine].Status.Error OR 
   arrAxisCtrl[AxiseNo.AxisName.AnCarryingWhirling].Status.Error OR
   arrAxisCtrl[AxiseNo.AxisName.AndeviationX1].Status.Error OR 
   arrAxisCtrl[AxiseNo.AxisName.AndeviationX2].Status.Error OR
   arrAxisCtrl[AxiseNo.AxisName.AndeviationY].Status.Error THEN
	An_Gohoming:=FALSE;//正极取片回原点中
		Step_InitAnDT:=9999;	
END_IF		

				
35://正极送片搬运升降、正极叠片搬运升降轴回原点
	arrAxisCtrl[AxiseNo.AxisName.AnCarryingUpDown].Cmd.bHome:=TRUE;//正极送片搬运轴回原点
	arrAxisCtrl[AxiseNo.AxisName.AnDTCarryingUpDown].Cmd.bHome:=TRUE;//正极叠片搬运回原点
	Step_InitAnDT:=40;
	
40://判断回原点是否完成
	IF NOT An_GohomeTon.Q THEN
			An_GohomeTon.IN:=TRUE;
	ELSE		
				IF arrAxisCtrl[AxiseNo.AxisName.AnCarryingUpDown].Status.Homed AND arrAxisCtrl[AxiseNo.AxisName.AnDTCarryingUpDown].Status.Homed  AND 
					arrAxisCtrl[AxiseNo.AxisName.AnCarryingUpDown].Status.NoMoving AND arrAxisCtrl[AxiseNo.AxisName.AnDTCarryingUpDown].Status.NoMoving  THEN
					arrAxisCtrl[AxiseNo.AxisName.AnCarryingUpDown].Cmd.bHome:=FALSE;//正极送片搬运轴回原点
					arrAxisCtrl[AxiseNo.AxisName.AnDTCarryingUpDown].Cmd.bHome:=FALSE;//正极叠片搬运回原点
					An_GohomeTon.IN:=FALSE;
					Step_InitAnDT:=45;
				ELSIF  arrAxisCtrl[AxiseNo.AxisName.AnCarryingUpDown].Status.Error OR arrAxisCtrl[AxiseNo.AxisName.AnDTCarryingUpDown].Status.Error THEN
						arrAxisCtrl[AxiseNo.AxisName.AnCarryingUpDown].Cmd.bHome:=FALSE;//正极送片搬运轴回原点
						arrAxisCtrl[AxiseNo.AxisName.AnDTCarryingUpDown].Cmd.bHome:=FALSE;//正极叠片搬运回原点
						An_GohomeTon.IN:=FALSE;
						An_Gohoming:=FALSE;//正极取片回原点中
						Step_InitAnDT:=9999;	  
				END_IF
	END_IF
45:
	IF arrAxisCtrl[AxiseNo.AxisName.AnDTCarryingUpDown].Status.Homed AND arrAxisCtrl[AxiseNo.AxisName.AnDTCarryingUpDown].Status.NoMoving THEN
		IF arrAxisCtrl[AxiseNo.AxisName.AnDTCarryingUpDown].Cmd.arrbRealPoint[5]  THEN
			arrAxisCtrl[AxiseNo.AxisName.AnDTCarryingUpDown].Cmd.iGoSetPos:=0;
			Step_InitAnDT:=50;
		ELSE
		   arrAxisCtrl[AxiseNo.AxisName.AnDTCarryingUpDown].Cmd.iGoSetPos:=5;
		END_IF	
	END_IF		
	IF  arrAxisCtrl[AxiseNo.AxisName.AnDTCarryingUpDown].Status.Error THEN
		An_Gohoming:=FALSE;//正极取片回原点中
		Step_InitAnDT:=9999;
	END_IF		
	
50://NG料盒气缸伸出
IF arrAxisCtrl[AxiseNo.AxisName.AnDTCarryingUpDown].Cmd.arrbRealPoint[5] OR arrCyCtrl[arrCyNo.CylinderName.AnScrapbinCy].Io.DIOnSwitch THEN
	arrCyCtrl[arrCyNo.CylinderName.AnScrapbinCy].Cmd.bON:=TRUE;//正极纠偏气缸伸出
	IF  arrCyCtrl[arrCyNo.CylinderName.AnScrapbinCy].Status.ONState THEN
		Step_InitAnDT:=60;	
	ELSIF arrCyCtrl[arrCyNo.CylinderName.AnScrapbinCy].Status.Error1 OR  arrCyCtrl[arrCyNo.CylinderName.AnScrapbinCy].Status.Error2 THEN
		An_Gohoming:=FALSE;//正极取片回原点中
		Step_InitAnDT:=9999;
	END_IF	
ELSE
	Mach_Control.An_b.Error[41] :=TRUE;//正极机械手初始化时，叠台搬运升降不在避让位
	An_Gohoming:=FALSE;//正极取片回原点中
	Step_InitAnDT:=9999;
END_IF	
	
60://正极送片搬运平移、叠片搬运平移、送片搬运旋转轴回原点、正极纠偏X1、正极纠偏X2、正极纠偏Y回原点
	arrAxisCtrl[AxiseNo.AxisName.AnCarryingLine].Cmd.bHome:=TRUE;//正极送片搬运平移轴回原点
	//arrAxisCtrl[AxiseNo.AxisName.AnCarryingWhirling].Cmd.bHome:=TRUE;//正极送片搬运旋转轴回原点								
	arrAxisCtrl[AxiseNo.AxisName.AndeviationX1].Cmd.bHome:=TRUE;//正极纠偏X1
	arrAxisCtrl[AxiseNo.AxisName.AndeviationX2].Cmd.bHome:=TRUE;//正极纠偏X2				
	arrAxisCtrl[AxiseNo.AxisName.AndeviationY].Cmd.bHome:=TRUE;//正极纠偏Y	
	An_CarryingTorMark:=TRUE;//正极搬运1移位力矩判断标志位									
	Step_InitAnDT:=70;
70://判断正极送片搬运平移、叠片搬运平移、送片搬运旋转回原点是否完成
	IF NOT An_GohomeTon.Q THEN		
		An_GohomeTon.IN:=TRUE;
	ELSE		
		IF arrAxisCtrl[AxiseNo.AxisName.AnCarryingLine].Status.Homed AND arrAxisCtrl[AxiseNo.AxisName.AnCarryingLine].Status.NoMoving (*AND
		 arrAxisCtrl[AxiseNo.AxisName.AnCarryingWhirling].Status.Homed*) AND  arrAxisCtrl[AxiseNo.AxisName.AnCarryingWhirling].Status.NoMoving  AND   						
		arrAxisCtrl[AxiseNo.AxisName.AndeviationX1].Status.Homed AND arrAxisCtrl[AxiseNo.AxisName.AndeviationX1].Status.NoMoving AND 
		arrAxisCtrl[AxiseNo.AxisName.AndeviationX2].Status.Homed AND arrAxisCtrl[AxiseNo.AxisName.AndeviationX2].Status.NoMoving AND
			arrAxisCtrl[AxiseNo.AxisName.AndeviationY].Status.Homed AND arrAxisCtrl[AxiseNo.AxisName.AndeviationY].Status.NoMoving   THEN
			arrAxisCtrl[AxiseNo.AxisName.AnCarryingLine].Cmd.bHome:=FALSE;//正极送片搬运平移轴回原点
			arrAxisCtrl[AxiseNo.AxisName.AnDTCarryingLine].Cmd.bHome:=FALSE;//正极叠片搬运平移轴回原点
			arrAxisCtrl[AxiseNo.AxisName.AnCarryingWhirling].Cmd.bHome:=FALSE;//正极送片搬运旋转轴回原点		
			arrAxisCtrl[AxiseNo.AxisName.AndeviationX1].Cmd.bHome:=FALSE;//正极纠偏X1		
			arrAxisCtrl[AxiseNo.AxisName.AndeviationX2].Cmd.bHome:=FALSE;//正极纠偏X2
			arrAxisCtrl[AxiseNo.AxisName.AndeviationY].Cmd.bHome:=FALSE;//正极纠偏Y
			An_CarryingTorMark:=FALSE;//正极搬运1移位力矩判断标志位			
			An_GohomeTon.IN:=FALSE;
			Step_InitAnDT:=75;
		ELSIF arrAxisCtrl[AxiseNo.AxisName.AnCarryingLine].Status.Error OR arrAxisCtrl[AxiseNo.AxisName.AnCarryingWhirling].Status.Error OR				
			arrAxisCtrl[AxiseNo.AxisName.AndeviationX1].Status.Error OR arrAxisCtrl[AxiseNo.AxisName.AndeviationX2].Status.Error OR 
			arrAxisCtrl[AxiseNo.AxisName.AndeviationY].Status.Error THEN
			arrAxisCtrl[AxiseNo.AxisName.AnCarryingLine].Cmd.bHome:=FALSE;//正极送片搬运平移轴回原点
			arrAxisCtrl[AxiseNo.AxisName.AnDTCarryingLine].Cmd.bHome:=FALSE;//正极叠片搬运平移轴回原点
			arrAxisCtrl[AxiseNo.AxisName.AnCarryingWhirling].Cmd.bHome:=FALSE;//正极送片搬运旋转轴回原点		
			arrAxisCtrl[AxiseNo.AxisName.AndeviationX1].Cmd.bHome:=FALSE;//正极纠偏X1		
			arrAxisCtrl[AxiseNo.AxisName.AndeviationX2].Cmd.bHome:=FALSE;//正极纠偏X2
			arrAxisCtrl[AxiseNo.AxisName.AndeviationY].Cmd.bHome:=FALSE;//正极纠偏Y
			An_GohomeTon.IN:=FALSE;
			An_Gohoming:=FALSE;//正极取片回原点中
			Step_InitAnDT:=9999;
		END_IF
	END_IF
75:
	//极送片搬运平移轴移动至初始位
	IF arrAxisCtrl[AxiseNo.AxisName.AnCarryingLine].Status.Homed AND arrAxisCtrl[AxiseNo.AxisName.AnCarryingLine].Status.NoMoving THEN
		IF arrAxisCtrl[AxiseNo.AxisName.AnCarryingLine].Cmd.arrbRealPoint[1] THEN
		   arrAxisCtrl[AxiseNo.AxisName.AnCarryingLine].Cmd.iGoSetPos:=0;
		 ELSE
			arrAxisCtrl[AxiseNo.AxisName.AnCarryingLine].Cmd.iGoSetPos:=1; 
		END_IF	
	END_IF
	(*//正极送片搬运旋转轴移动至初始位
	IF arrAxisCtrl[AxiseNo.AxisName.AnCarryingWhirling].Status.Homed AND arrAxisCtrl[AxiseNo.AxisName.AnCarryingWhirling].Status.NoMoving THEN
		IF arrAxisCtrl[AxiseNo.AxisName.AnCarryingWhirling].Cmd.arrbRealPoint[1]  THEN
			arrAxisCtrl[AxiseNo.AxisName.AnCarryingWhirling].Cmd.iGoSetPos:=0;
		ELSE
		   arrAxisCtrl[AxiseNo.AxisName.AnCarryingWhirling].Cmd.iGoSetPos:=1;
		END_IF
	END_IF*)
	//正极纠偏X1
	IF arrAxisCtrl[AxiseNo.AxisName.AndeviationX1].Status.Homed AND arrAxisCtrl[AxiseNo.AxisName.AndeviationX1].Status.NoMoving THEN
		IF arrAxisCtrl[AxiseNo.AxisName.AndeviationX1].Cmd.arrbRealPoint[1]  THEN
			arrAxisCtrl[AxiseNo.AxisName.AndeviationX1].Cmd.iGoSetPos:=0;
		ELSE
		   arrAxisCtrl[AxiseNo.AxisName.AndeviationX1].Cmd.iGoSetPos:=1;
		END_IF
	END_IF
	//正极纠偏X2
	IF arrAxisCtrl[AxiseNo.AxisName.AndeviationX2].Status.Homed AND arrAxisCtrl[AxiseNo.AxisName.AndeviationX2].Status.NoMoving THEN
		IF arrAxisCtrl[AxiseNo.AxisName.AndeviationX2].Cmd.arrbRealPoint[1]  THEN
			arrAxisCtrl[AxiseNo.AxisName.AndeviationX2].Cmd.iGoSetPos:=0;
		ELSE
		   arrAxisCtrl[AxiseNo.AxisName.AndeviationX2].Cmd.iGoSetPos:=1;
		END_IF
	END_IF	
	//正极纠偏Y
	IF arrAxisCtrl[AxiseNo.AxisName.AndeviationY].Status.Homed AND arrAxisCtrl[AxiseNo.AxisName.AndeviationY].Status.NoMoving THEN
		IF arrAxisCtrl[AxiseNo.AxisName.AndeviationY].Cmd.arrbRealPoint[1]  THEN
			arrAxisCtrl[AxiseNo.AxisName.AndeviationY].Cmd.iGoSetPos:=0;
		ELSE
		   arrAxisCtrl[AxiseNo.AxisName.AndeviationY].Cmd.iGoSetPos:=1;
		END_IF
	END_IF								
	
	IF 	arrAxisCtrl[AxiseNo.AxisName.AnCarryingLine].Cmd.arrbRealPoint[1] AND arrAxisCtrl[AxiseNo.AxisName.AnCarryingLine].Status.NoMoving AND
		(*arrAxisCtrl[AxiseNo.AxisName.AnCarryingWhirling].Cmd.arrbRealPoint[1] AND *)arrAxisCtrl[AxiseNo.AxisName.AnCarryingWhirling].Status.NoMoving AND
		arrAxisCtrl[AxiseNo.AxisName.AndeviationX1].Cmd.arrbRealPoint[1]  AND arrAxisCtrl[AxiseNo.AxisName.AndeviationX1].Status.NoMoving AND
		arrAxisCtrl[AxiseNo.AxisName.AndeviationX2].Cmd.arrbRealPoint[1] AND arrAxisCtrl[AxiseNo.AxisName.AndeviationX2].Status.NoMoving AND
		arrAxisCtrl[AxiseNo.AxisName.AndeviationY].Cmd.arrbRealPoint[1]	 AND	arrAxisCtrl[AxiseNo.AxisName.AndeviationY].Status.NoMoving THEN
					Step_InitAnDT:=80;
					arrAxisCtrl[AxiseNo.AxisName.AnCarryingWhirling].Cmd.bHome:=TRUE;//正极送片搬运旋转轴回原点
					
	ELSIF  arrAxisCtrl[AxiseNo.AxisName.AnCarryingLine].Status.Error AND arrAxisCtrl[AxiseNo.AxisName.AnCarryingWhirling].Status.Error AND
		arrAxisCtrl[AxiseNo.AxisName.AndeviationX1].Status.Error AND arrAxisCtrl[AxiseNo.AxisName.AndeviationX2].Status.Error AND 
		arrAxisCtrl[AxiseNo.AxisName.AndeviationY].Status.Error THEN
		An_Gohoming:=FALSE;//正极取片回原点中
		Step_InitAnDT:=9999;
	END_IF	
80://正极送片搬运旋转轴回原点	
IF  arrAxisCtrl[AxiseNo.AxisName.AnCarryingWhirling].Status.Homed		THEN
	arrAxisCtrl[AxiseNo.AxisName.AnCarryingWhirling].Cmd.bHome:=FALSE;//正极送片搬运旋转轴回原点	
	Step_InitAnDT:=83;	
END_IF			

83://正极送片搬运旋转轴移动至初始位
	IF arrAxisCtrl[AxiseNo.AxisName.AnCarryingWhirling].Status.Homed AND arrAxisCtrl[AxiseNo.AxisName.AnCarryingWhirling].Status.NoMoving THEN
		IF arrAxisCtrl[AxiseNo.AxisName.AnCarryingWhirling].Cmd.arrbRealPoint[1]  THEN
			arrAxisCtrl[AxiseNo.AxisName.AnCarryingWhirling].Cmd.iGoSetPos:=0;
			Step_InitAnDT:=85;
		ELSE
		   arrAxisCtrl[AxiseNo.AxisName.AnCarryingWhirling].Cmd.iGoSetPos:=1;
		END_IF
	END_IF

85://叠片搬运回原点							
	arrAxisCtrl[AxiseNo.AxisName.AnDTCarryingLine].Cmd.bHome:=TRUE;//正极叠片搬运平移轴回原点
	An_DTCarryingTorMark:=TRUE;//正极叠台搬运力矩判断标志位	
	Step_InitAnDT:=90;	
90://判断叠片搬运回原点是否完成
	IF NOT An_GohomeTon.Q THEN
		An_GohomeTon.IN:=TRUE;
	ELSE
		IF arrAxisCtrl[AxiseNo.AxisName.AnDTCarryingLine].Status.Homed AND arrAxisCtrl[AxiseNo.AxisName.AnDTCarryingLine].Status.NoMoving  THEN
			An_GohomeTon.IN:=FALSE;	
			arrAxisCtrl[AxiseNo.AxisName.AnDTCarryingLine].Cmd.bHome:=FALSE;//正极叠片搬运平移轴回原点
			An_DTCarryingTorMark:=FALSE;//正极叠台搬运力矩判断标志位	
			Step_InitAnDT:=100;
		ELSIF arrAxisCtrl[AxiseNo.AxisName.AnDTCarryingLine].Status.Error THEN
			An_GohomeTon.IN:=FALSE;	
			arrAxisCtrl[AxiseNo.AxisName.AnDTCarryingLine].Cmd.bHome:=FALSE;//正极叠片搬运平移轴回原点
		    An_Gohoming:=FALSE;//正极取片回原点中
			Step_InitAnDT:=9999;
		END_IF
	END_IF
100://轴移动到初始位置	
	//正极叠片搬运平移轴移动至初始位
	IF arrAxisCtrl[AxiseNo.AxisName.AnDTCarryingLine].Status.Homed AND arrAxisCtrl[AxiseNo.AxisName.AnDTCarryingLine].Status.NoMoving THEN
		IF arrAxisCtrl[AxiseNo.AxisName.AnDTCarryingLine].Cmd.arrbRealPoint[1]  THEN
			arrAxisCtrl[AxiseNo.AxisName.AnDTCarryingLine].Cmd.iGoSetPos:=0;
			Step_InitAnDT:=110;
		ELSE
		   arrAxisCtrl[AxiseNo.AxisName.AnDTCarryingLine].Cmd.iGoSetPos:=1;
		END_IF	
	ELSIF arrAxisCtrl[AxiseNo.AxisName.AnDTCarryingLine].Status.Error THEN
		An_Gohoming:=FALSE;//正极取片回原点中
		Step_InitAnDT:=9999;
	END_IF
110:
	arrCyCtrl[arrCyNo.ElectValveName.AnCarryingVacuum].Cmd.bOFF:=TRUE;//正极搬运升降取料真空关
	arrCyCtrl[arrCyNo.ElectValveName.AnCarryingVacuum].Cmd.bON:=FALSE;//正极搬运升降取料真空关
	
	arrCyCtrl[arrCyNo.ElectValveName.AnCarryingVacuumBark].Cmd.bOFF:=TRUE;//正极搬运升降取料破真空关
	arrCyCtrl[arrCyNo.ElectValveName.AnCarryingVacuumBark].Cmd.bON:=FALSE;//正极搬运升降取料破真空关
	
	arrCyCtrl[arrCyNo.ElectValveName.AndeviationVacuum].Cmd.bOFF:=TRUE;//正极纠偏平台真空关
	arrCyCtrl[arrCyNo.ElectValveName.AndeviationVacuum].Cmd.bON:=FALSE;//正极纠偏平台真空关
	
	arrCyCtrl[arrCyNo.ElectValveName.AndeviationVacuumBark].Cmd.bOFF:=TRUE;//正极纠偏平台破真空关
	arrCyCtrl[arrCyNo.ElectValveName.AndeviationVacuumBark].Cmd.bON:=FALSE;//正极纠偏平台破真空关
	
	arrCyCtrl[arrCyNo.ElectValveName.AnDTCarryingVacuum].Cmd.bOFF:=FALSE;//正极叠片搬运真空关
	arrCyCtrl[arrCyNo.ElectValveName.AnDTCarryingVacuum].Cmd.bON:=TRUE;//正极叠片搬运真空关
	
	arrCyCtrl[arrCyNo.ElectValveName.AnDTCarryingVacuumBark].Cmd.bON:=TRUE;//正极叠片搬运破真空关	
	arrCyCtrl[arrCyNo.ElectValveName.AnDTCarryingVacuumBark].Cmd.bOFF:=FALSE;//正极叠片搬运破真空关				
	//正极送片搬运升降移动至等待位
	IF arrAxisCtrl[AxiseNo.AxisName.AnCarryingUpDown].Status.Homed AND arrAxisCtrl[AxiseNo.AxisName.AnCarryingUpDown].Status.NoMoving THEN
		IF arrAxisCtrl[AxiseNo.AxisName.AnCarryingUpDown].Cmd.arrbRealPoint[4] THEN
		   arrAxisCtrl[AxiseNo.AxisName.AnCarryingUpDown].Cmd.iGoSetPos:=0;
		 ELSE
			arrAxisCtrl[AxiseNo.AxisName.AnCarryingUpDown].Cmd.iGoSetPos:=4;
		END_IF
	END_IF
	//正极叠片搬运升降移动至等待位
	IF arrAxisCtrl[AxiseNo.AxisName.AnDTCarryingUpDown].Status.Homed AND arrAxisCtrl[AxiseNo.AxisName.AnDTCarryingUpDown].Status.NoMoving THEN
		IF  arrAxisCtrl[AxiseNo.AxisName.AnDTCarryingUpDown].Cmd.arrbRealPoint[4] THEN
				arrAxisCtrl[AxiseNo.AxisName.AnDTCarryingUpDown].Cmd.iGoSetPos:=0;
		 ELSE
				arrAxisCtrl[AxiseNo.AxisName.AnDTCarryingUpDown].Cmd.iGoSetPos:=4;
		END_IF	
	END_IF		
	IF  	arrAxisCtrl[AxiseNo.AxisName.AnCarryingUpDown].Cmd.arrbRealPoint[4] AND arrAxisCtrl[AxiseNo.AxisName.AnCarryingUpDown].Status.NoMoving  AND 
		arrAxisCtrl[AxiseNo.AxisName.AnDTCarryingUpDown].Cmd.arrbRealPoint[4] AND 	arrAxisCtrl[AxiseNo.AxisName.AnDTCarryingUpDown].Status.NoMoving  THEN
		An_GohomeDone:=TRUE;//正极回原点完成
		An_Gohoming:=FALSE;//正极取片回原点中
		Step_InitAnDT:=0;
	ELSIF arrAxisCtrl[AxiseNo.AxisName.AnCarryingUpDown].Status.Error OR arrAxisCtrl[AxiseNo.AxisName.AnDTCarryingUpDown].Status.Error THEN
		An_Gohoming:=FALSE;//正极取片回原点中
		Step_InitAnDT:=9999;
	END_IF
END_CASE
END_IF
END_ACTION

ACTION An_OverNG:
DT_TON[1](IN:= , PT:=T#300MS , Q=> , ET=> );//
DT_TON[2](IN:= , PT:=T#300MS , Q=> , ET=> );//
DT_TON[3](IN:= , PT:=T#200MS , Q=> , ET=> );//
DT_TON[4](IN:= , PT:=T#200MS , Q=> , ET=> );//
(*******************************************************************************************************踢正极对齐度NG片**************************************************************************************************************************)
 IF   An_OverNGStep=1630 THEN
	arrAxisCtrl[AxiseNo.AxisName.AnDTCarryingUpDown].Cmd.fOverride:=50;
 ELSE
   arrAxisCtrl[AxiseNo.AxisName.AnDTCarryingUpDown].Cmd.fOverride:=100;
 END_IF
 

 
 IF  AnOverNGcount>=3 OR CaOverNGcount>=3 THEN
     OversequelNG:=TRUE;	
 END_IF
 
IF Mach_Control.U.DT_iMode=1 THEN//在自动状态下
   CASE An_OverNGStep OF   
			1000://判断正极叠台搬运是否有片，有片的话放到纠偏台
						fAnScaling:=1;//20240508 CF
		            	fCaScaling:=1;//20240508 CF		
						AnOverNGcount:=AnOverNGcount+1;
						IF arrCyCtrl[arrCyNo.ElectValveName.AnDTCarryingVacuum].Io.DIOnSwitch AND  Mach_Control.An_b.An_DPCarryingFalg  THEN//正极再取片位且叠台搬运有片,把当前片放到纠偏台
							An_OverNGStep:=1010;
						ELSE
							An_OverNGStep:=1050;	
						END_IF
	
			1010://纠偏台回初始位
				//纠偏平台X1移动至初始位
				IF NOT DP_SinStepe THEN
					IF arrAxisCtrl[AxiseNo.AxisName.AndeviationX1].Status.Homed  AND arrAxisCtrl[AxiseNo.AxisName.AndeviationX1].Status.NoMoving AND NOT  arrAxisCtrl[AxiseNo.AxisName.AndeviationX1].Status.Error THEN
						IF arrAxisCtrl[AxiseNo.AxisName.AndeviationX1].Cmd.arrbRealPoint[1] THEN
							arrAxisCtrl[AxiseNo.AxisName.AndeviationX1].Cmd.iGoSetPos:=0;
						ELSE
							arrAxisCtrl[AxiseNo.AxisName.AndeviationX1].Cmd.iGoSetPos:=1;
						END_IF					
					END_IF
					//纠偏平台X2移动至初始位
					IF arrAxisCtrl[AxiseNo.AxisName.AndeviationX2].Status.Homed  AND arrAxisCtrl[AxiseNo.AxisName.AndeviationX2].Status.NoMoving AND NOT  arrAxisCtrl[AxiseNo.AxisName.AndeviationX2].Status.Error THEN
						IF arrAxisCtrl[AxiseNo.AxisName.AndeviationX2].Cmd.arrbRealPoint[1] THEN
							arrAxisCtrl[AxiseNo.AxisName.AndeviationX2].Cmd.iGoSetPos:=0;
						ELSE
							arrAxisCtrl[AxiseNo.AxisName.AndeviationX2].Cmd.iGoSetPos:=1;
						END_IF					
					END_IF
					//纠偏平台X2移动至初始位
					IF arrAxisCtrl[AxiseNo.AxisName.AndeviationY].Status.Homed  AND arrAxisCtrl[AxiseNo.AxisName.AndeviationY].Status.NoMoving AND NOT  arrAxisCtrl[AxiseNo.AxisName.AndeviationY].Status.Error THEN
						IF arrAxisCtrl[AxiseNo.AxisName.AndeviationY].Cmd.arrbRealPoint[1] THEN
							arrAxisCtrl[AxiseNo.AxisName.AndeviationY].Cmd.iGoSetPos:=0;
						ELSE
							arrAxisCtrl[AxiseNo.AxisName.AndeviationY].Cmd.iGoSetPos:=1;
						END_IF					
					END_IF
					IF arrAxisCtrl[AxiseNo.AxisName.AndeviationX1].Cmd.arrbRealPoint[1] AND arrAxisCtrl[AxiseNo.AxisName.AndeviationX2].Cmd.arrbRealPoint[1] AND arrAxisCtrl[AxiseNo.AxisName.AndeviationY].Cmd.arrbRealPoint[1] THEN
						DT_SingeMode();//单步选择	
						An_OverNGStep:=1020;
                        DT_TON[3].IN:=FALSE; 	
					END_IF	
				END_IF
			1020://叠台搬运极片放回纠偏台
				IF NOT DP_SinStepe THEN
					IF arrAxisCtrl[AxiseNo.AxisName.AnDTCarryingLine].Cmd.arrbRealPoint[1]  AND NOT Mach_Control.An_b.An_deviationFalg THEN 
						IF arrAxisCtrl[AxiseNo.AxisName.AnDTCarryingUpDown].Cmd.arrbRealPoint[2] THEN
							arrAxisCtrl[AxiseNo.AxisName.AnDTCarryingUpDown].Cmd.iGoSetPos:=0;
					    ELSE
							arrAxisCtrl[AxiseNo.AxisName.AnDTCarryingUpDown].Cmd.iGoSetPos:=2;//正极叠台搬运下降至取片位
					    END_IF
                   END_IF
				       IF arrAxisCtrl[AxiseNo.AxisName.AnDTCarryingUpDown].Cmd.arrbRealPoint[2] THEN
				           	/// 吸盘破真空    纠偏台开真空
				
							arrCyCtrl[arrCyNo.ElectValveName.AnDTCarryingVacuum].Cmd.bOFF:=FALSE;//正极叠片搬运升降真空关
							arrCyCtrl[arrCyNo.ElectValveName.AnDTCarryingVacuum].Cmd.bON:=TRUE;//正极叠片搬运升降真空关
						
							arrCyCtrl[arrCyNo.ElectValveName.AndeviationVacuum].Cmd.bON:=TRUE;	//正极纠偏台真空			
							arrCyCtrl[arrCyNo.ElectValveName.AndeviationVacuum].Cmd.bOFF:=FALSE;	//正极纠偏台真空	   
							DT_SingeMode();//单步选择	
							An_OverNGStep:=1030;
							DT_TON[3].IN:=TRUE;
							Mach_Control.An_b.An_deviationFalg:=TRUE;//置位纠偏平台有料标记
						    Mach_Control.An_b.An_DPCarryingFalg:=FALSE;//正极搬运真空吸盘有料标记复位
	                    END_IF
				END_IF
			1030://叠台搬运极片上升至凸轮耦合初始高度
				IF NOT DP_SinStepe  AND DT_TON[3].Q THEN
					IF arrAxisCtrl[AxiseNo.AxisName.AnDTCarryingUpDown].Cmd.arrbRealPoint[4]  THEN
						arrAxisCtrl[AxiseNo.AxisName.AnDTCarryingUpDown].Cmd.iGoSetPos:=0;
						/// 吸盘破真空    纠偏台开真空
						Mach_Control.An_b.An_deviationFalg:=TRUE;//置位纠偏平台有料标记
						Mach_Control.An_b.An_DPCarryingFalg:=FALSE;//正极搬运真空吸盘有料标记复位
						Par.stDT_date.An_MQ_Slice[1]:=Par.stDT_date.An_MQ_Slice[2];
						DT_SingeMode();//单步选择	
						An_OverNGStep:=1050;
						DT_TON[3].IN:=FALSE;
					ELSE
						arrAxisCtrl[AxiseNo.AxisName.AnDTCarryingUpDown].Cmd.iGoSetPos:=4;//正极搬运升降2上升至凸轮耦合初始高度
					END_IF			
				END_IF		   
		
            1050://判断主轴是否停止、是否在初始位、是否有轴在耦合中
					IF NOT DP_SinStepe THEN
								IF arrAxis[AxiseNo.VirAxisName.VirMain].Status.NotMoving AND arrAxis[AxiseNo.VirAxisName.VirMain].NcToPlc.SetPos=0 AND NOT DT_AxiseCoupling THEN
									DT_SingeMode();//单步选择
									An_OverNGStep:=1070;
								ELSE
									DP_Step1:=100;//调用主轴回初始位子程序
									DT_SingeMode();//单步选择
									An_OverNGStep:=1060;
								END_IF
			    	END_IF		
			1060://判断主轴的模长的当前位置是否为0
				IF NOT DP_SinStepe THEN
					IF DP_Step1=6666 AND arrAxis[AxiseNo.VirAxisName.VirMain].Status.NotMoving AND arrAxis[AxiseNo.VirAxisName.VirMain].NcToPlc.SetPos=0 AND NOT DT_AxiseCoupling  THEN
						DT_SingeMode();//单步选择
						An_OverNGStep:=1070;
					END_IF	
				END_IF							

			1070://判断NG气缸是否在安全位
					IF arrCyCtrl[arrCyNo.CylinderName.AnScrapbinCy].Status.ONState AND arrCyCtrl[arrCyNo.CylinderName.CaScrapbinUDCy].Status.OFFState AND
						arrCyCtrl[arrCyNo.CylinderName.AnScrapbinCy].Status.ONState AND arrCyCtrl[arrCyNo.CylinderName.PreDiaph].Status.OFFState AND 
						arrCyCtrl[arrCyNo.CylinderName.PoleHotCutterCy].Status.OFFState AND arrCyCtrl[arrCyNo.CylinderName.PoleTapeCy].Status.OFFState AND
						arrCyCtrl[arrCyNo.CylinderName.PoleTapeSplicerRCy].Status.ONState AND arrCyCtrl[arrCyNo.CylinderName.PoleTapeSplicerLCy].Status.ONState AND 
                        arrAxisCtrl[AxiseNo.AxisName.LeftYDUpDown].Cmd.arrbRealPoint[1] AND arrAxisCtrl[AxiseNo.AxisName.RightYDUpDown].Cmd.arrbRealPoint[1]    THEN
						An_OverNGStep:=1100;		
					ELSE
						An_OverNGStep:=1080;	
					END_IF
			1080:
						arrCyCtrl[arrCyNo.CylinderName.AnScrapbinCy].Cmd.bON:=TRUE;
						arrCyCtrl[arrCyNo.CylinderName.PreDiaph].Cmd.bOFF:=TRUE;
						arrCyCtrl[arrCyNo.CylinderName.PoleHotCutterCy].Cmd.bOFF:=TRUE;
						arrCyCtrl[arrCyNo.CylinderName.PoleTapeCy].Cmd.bOFF:=TRUE;
						arrCyCtrl[arrCyNo.CylinderName.PoleTapeSplicerRCy].Cmd.bON:=TRUE;
						arrCyCtrl[arrCyNo.CylinderName.PoleTapeSplicerLCy].Cmd.bON:=TRUE;
						arrCyCtrl[arrCyNo.CylinderName.AnScrapbinCy].Cmd.bON:=TRUE;
						IF   arrCyCtrl[arrCyNo.CylinderName.AnScrapbinCy].Status.ONState AND  arrCyCtrl[arrCyNo.CylinderName.PreDiaph].Status.OFFState AND 
							arrCyCtrl[arrCyNo.CylinderName.PoleHotCutterCy].Status.OFFState AND arrCyCtrl[arrCyNo.CylinderName.PoleTapeCy].Status.OFFState AND
							arrCyCtrl[arrCyNo.CylinderName.PoleTapeSplicerRCy].Status.ONState AND arrCyCtrl[arrCyNo.CylinderName.PoleTapeSplicerLCy].Status.ONState THEN
							An_OverNGStep:=1090;									
						END_IF
			1090:
					arrCyCtrl[arrCyNo.CylinderName.CaScrapbinUDCy].Cmd.bOFF:=TRUE;
					IF  arrCyCtrl[arrCyNo.CylinderName.CaScrapbinUDCy].Status.OFFState AND  arrAxisCtrl[AxiseNo.AxisName.LeftYDUpDown].Cmd.arrbRealPoint[1] 
                         AND arrAxisCtrl[AxiseNo.AxisName.RightYDUpDown].Cmd.arrbRealPoint[1] THEN
						An_OverNGStep:=1100;	
					END_IF	

              1100:
						IF NOT DP_SinStepe AND TailCurlSEPTA_SafePos THEN		
									Scan_TON[2].IN:=TRUE;	
										IF 	An_CarryingPos1  THEN//正极搬运、叠片各轴在初始位
											         Scan_TON[1].IN:=TRUE;	
													 DTPosError[11]:=FALSE;
													 IF CA_CarryingPos2  THEN//负极在叠片位	
														             DTPosError[12]:=FALSE;
																IF arrAxisCtrl[AxiseNo.AxisName.SEPTATLine].Cmd.arrbRealPoint[1]   THEN													
																	DT_SingeMode();//单步选择											
																	An_OverNGStep:=1200;//													
																ELSE
																	Mach_Control.DT_b.Error[6]:=TRUE;//叠正极片凸轮耦合时，隔膜平移轴即不在正极叠片位，也不在正极叠片位报警
																//	An_OverNGStep:=9991;	
																END_IF;
													ELSIF CA_CarryingPos1  THEN//负极在取片位	
                                                                  DTPosError[12]:=FALSE;																	
																IF arrAxisCtrl[AxiseNo.AxisName.SEPTATLine].Cmd.arrbRealPoint[2]  THEN
																	DT_SingeMode();//单步选择										
																	An_OverNGStep:=1300;//
																ELSIF arrAxisCtrl[AxiseNo.AxisName.SEPTATLine].Cmd.arrbRealPoint[1] THEN
																	DT_SingeMode();//单步选择										
																	An_OverNGStep:=1400;//
																ELSE
																	Mach_Control.DT_b.Error[6]:=TRUE;//叠正极片凸轮耦合时，隔膜平移轴即不在正极叠片位，也不在正极叠片位报警
																	//An_OverNGStep:=9992;	
																END_IF;							
													ELSIF Scan_TON[1].Q THEN
																Scan_TON[1].IN:=FALSE;	
																//An_OverNGStep:=9993;
															   DTPosError[12]:=TRUE;
													END_IF
							    	ELSE
											IF (Ca_Step0=0 OR Ca_Step0=6666) AND (Ca_Step3=0 OR Ca_Step3=6666) AND Scan_TON[2].Q THEN
												Scan_TON[2].IN:=FALSE;		
												//An_OverNGStep:=9994;
												DTPosError[11]:=TRUE;
											END_IF
								END_IF
					END_IF		

              1600:	 //正极叠片升降移动至放片高度 		  
	           			IF NOT DP_SinStepe THEN					
									 IF arrAxisCtrl[AxiseNo.AxisName.AnDTCarryingUpDown].Status.Homed AND arrAxisCtrl[AxiseNo.AxisName.AnDTCarryingUpDown].Status.NoMoving AND 
										NOT arrAxisCtrl[AxiseNo.AxisName.AnDTCarryingUpDown].Status.Error AND arrAxisCtrl[AxiseNo.AxisName.AnDTCarryingLine].Cmd.arrbRealPoint[2] AND
                                             arrAxisCtrl[AxiseNo.AxisName.LeftYDUpDown].Cmd.arrbRealPoint[1] AND arrAxisCtrl[AxiseNo.AxisName.RightYDUpDown].Cmd.arrbRealPoint[1]       THEN
											IF arrAxisCtrl[AxiseNo.AxisName.AnDTCarryingUpDown].Cmd.arrbRealPoint[3] THEN
												arrAxisCtrl[AxiseNo.AxisName.AnDTCarryingUpDown].Cmd.iGoSetPos:=0;
											ELSE
												arrAxisCtrl[AxiseNo.AxisName.AnDTCarryingUpDown].Cmd.iGoSetPos:=3;//正极叠片升降移动至等待高度
											END_IF
									END_IF   	
								IF arrAxisCtrl[AxiseNo.AxisName.AnDTCarryingUpDown].Cmd.arrbRealPoint[3] THEN
								    DT_SingeMode();//单步选择
									An_OverNGStep:=1610;
								END_IF		
                       END_IF	   
		1610://	右刀升降轴上升至张开高度
						     arrCyCtrl[arrCyNo.ElectValveName.AnDTCarryingVacuum].Cmd.bOFF:=TRUE;//正极叠片搬运升降真空开
	                    	arrCyCtrl[arrCyNo.ElectValveName.AnDTCarryingVacuum].Cmd.bON:=FALSE;//正极叠片搬运升降真空开
						IF NOT DP_SinStepe THEN								
								IF 	arrAxisCtrl[AxiseNo.AxisName.RightYDUpDown].Status.Homed AND arrAxisCtrl[AxiseNo.AxisName.RightYDUpDown].Status.NoMoving THEN
									IF arrAxisCtrl[AxiseNo.AxisName.RightYDUpDown].Cmd.arrbRealPoint[15] THEN
										arrAxisCtrl[AxiseNo.AxisName.RightYDUpDown].Cmd.iGoSetPos:=0;
									ELSE
										arrAxisCtrl[AxiseNo.AxisName.RightYDUpDown].Cmd.iGoSetPos:=15;//右压刀升降上升至抽刀高度
									END_IF
								END_IF				
								IF arrAxisCtrl[AxiseNo.AxisName.RightYDUpDown].Cmd.arrbRealPoint[15] THEN
							     	DT_SingeMode();//单步选择
									An_OverNGStep:=1620;
								END_IF
						END_IF	   
	
            1620://	右压刀开合轴至张开位			   
					   IF NOT DP_SinStepe THEN
										IF 	arrAxisCtrl[AxiseNo.AxisName.RightYDLine].Status.Homed AND arrAxisCtrl[AxiseNo.AxisName.RightYDLine].Status.NoMoving THEN
												IF arrAxisCtrl[AxiseNo.AxisName.RightYDLine].Cmd.arrbRealPoint[2] THEN
													arrAxisCtrl[AxiseNo.AxisName.RightYDLine].Cmd.iGoSetPos:=0;
												ELSE
													arrAxisCtrl[AxiseNo.AxisName.RightYDLine].Cmd.iGoSetPos:=2;//右压刀开合至张开位	
												END_IF		
										END_IF;	
											IF arrAxisCtrl[AxiseNo.AxisName.RightYDLine].Cmd.arrbRealPoint[2] THEN
													DT_SingeMode();//单步选择
													An_OverNGStep:=1630;											
											END_IF
							END_IF;
				   
	
         1630:	 //正极叠片升降移动至a等待高度 		  
	           			IF NOT DP_SinStepe THEN					
								 IF arrAxisCtrl[AxiseNo.AxisName.AnDTCarryingUpDown].Status.Homed AND arrAxisCtrl[AxiseNo.AxisName.AnDTCarryingUpDown].Status.NoMoving AND 
									NOT arrAxisCtrl[AxiseNo.AxisName.AnDTCarryingUpDown].Status.Error AND arrAxisCtrl[AxiseNo.AxisName.AnDTCarryingLine].Cmd.arrbRealPoint[2] AND
										 arrAxisCtrl[AxiseNo.AxisName.LeftYDUpDown].Cmd.arrbRealPoint[1] AND arrAxisCtrl[AxiseNo.AxisName.RightYDLine].Cmd.arrbRealPoint[2]     THEN
										IF arrAxisCtrl[AxiseNo.AxisName.AnDTCarryingUpDown].Cmd.arrbRealPoint[4] THEN
											arrAxisCtrl[AxiseNo.AxisName.AnDTCarryingUpDown].Cmd.iGoSetPos:=0;
										ELSE
											arrAxisCtrl[AxiseNo.AxisName.AnDTCarryingUpDown].Cmd.iGoSetPos:=4;//正极叠片升降移动至等待高度
										END_IF
								END_IF 
                                (*
								IF 	arrAxisCtrl[AxiseNo.AxisName.RightYDUpDown].Status.Homed AND arrAxisCtrl[AxiseNo.AxisName.RightYDUpDown].Status.NoMoving THEN
									IF arrAxisCtrl[AxiseNo.AxisName.RightYDUpDown].Cmd.arrbRealPoint[1] THEN
										arrAxisCtrl[AxiseNo.AxisName.RightYDUpDown].Cmd.iGoSetPos:=0;
									ELSE
										arrAxisCtrl[AxiseNo.AxisName.RightYDUpDown].Cmd.iGoSetPos:=1;//右压刀升降上升至初始高度
									END_IF
								END_IF													
  	                            *)
								IF arrAxisCtrl[AxiseNo.AxisName.AnDTCarryingUpDown].Cmd.arrbRealPoint[4] AND arrAxisCtrl[AxiseNo.AxisName.RightYDUpDown].Cmd.arrbRealPoint[15] AND
                                    arrAxisCtrl[AxiseNo.AxisName.AnDTCarryingUpDown].Status.NoMoving  AND arrAxisCtrl[AxiseNo.AxisName.RightYDUpDown].Status.NoMoving    THEN
						         	DT_SingeMode();//单步选择
									An_OverNGStep:=1670;
								END_IF		
                       END_IF	   						
 (*
  		1640://	压刀升降上升至初始高度	
					IF NOT DP_SinStepe THEN								
								IF 	arrAxisCtrl[AxiseNo.AxisName.RightYDUpDown].Status.Homed AND arrAxisCtrl[AxiseNo.AxisName.RightYDUpDown].Status.NoMoving THEN
									IF arrAxisCtrl[AxiseNo.AxisName.RightYDUpDown].Cmd.arrbRealPoint[1] THEN
										arrAxisCtrl[AxiseNo.AxisName.RightYDUpDown].Cmd.iGoSetPos:=0;
									ELSE
										arrAxisCtrl[AxiseNo.AxisName.RightYDUpDown].Cmd.iGoSetPos:=1;//右压刀升降上升至初始高度
									END_IF
								END_IF				
								IF arrAxisCtrl[AxiseNo.AxisName.RightYDUpDown].Cmd.arrbRealPoint[1] THEN
							     	DT_SingeMode();//单步选择
									An_OverNGStep:=1641;
								END_IF
						END_IF	   
	
		1641://	右压刀开合移至初始位		
			       IF NOT DP_SinStepe THEN
								IF 	arrAxisCtrl[AxiseNo.AxisName.RightYDLine].Status.Homed AND arrAxisCtrl[AxiseNo.AxisName.RightYDLine].Status.NoMoving THEN
										IF arrAxisCtrl[AxiseNo.AxisName.RightYDLine].Cmd.arrbRealPoint[1] THEN
											arrAxisCtrl[AxiseNo.AxisName.RightYDLine].Cmd.iGoSetPos:=0;
											DT_SingeMode();//单步选择
											An_OverNGStep:=1650;
										ELSE
											arrAxisCtrl[AxiseNo.AxisName.RightYDLine].Cmd.iGoSetPos:=1;//右压刀开合至初始位
										END_IF		
                                END_IF;	
					END_IF;				
					
		   	1650://右压刀升降下降至初始位，压隔膜			
					  IF NOT DP_SinStepe THEN
	                         	IF 	arrAxisCtrl[AxiseNo.AxisName.RightYDUpDown].Status.Homed AND arrAxisCtrl[AxiseNo.AxisName.RightYDUpDown].Status.NoMoving THEN
										IF arrAxisCtrl[AxiseNo.AxisName.RightYDUpDown].Cmd.arrbRealPoint[1] THEN
											arrAxisCtrl[AxiseNo.AxisName.RightYDUpDown].Cmd.iGoSetPos:=0;
									     	DT_SingeMode();//单步选择
									    	An_OverNGStep:=1670;
										ELSE
											arrAxisCtrl[AxiseNo.AxisName.RightYDUpDown].Cmd.iGoSetPos:=1;//右压刀升降轴下降至初始高度
										END_IF
									END_IF							  
					  
					  END_IF					   
					   
		     //1660:	 //判断真空					   
	*)

           1670://判断主轴是否停止、是否在初始位、是否有轴在耦合中
					IF NOT DP_SinStepe THEN
								IF arrAxis[AxiseNo.VirAxisName.VirMain].Status.NotMoving AND arrAxis[AxiseNo.VirAxisName.VirMain].NcToPlc.SetPos=0 AND NOT DT_AxiseCoupling THEN
									DT_SingeMode();//单步选择
									An_OverNGStep:=1691;
								ELSE
									DP_Step1:=100;//调用主轴回初始位子程序
									DT_SingeMode();//单步选择
									An_OverNGStep:=1690;
								END_IF
			    	END_IF		
			1690://判断主轴的模长的当前位置是否为0
				IF NOT DP_SinStepe THEN
					IF DP_Step1=6666 AND arrAxis[AxiseNo.VirAxisName.VirMain].Status.NotMoving AND arrAxis[AxiseNo.VirAxisName.VirMain].NcToPlc.SetPos=0 AND NOT DT_AxiseCoupling  THEN
						DT_SingeMode();//单步选择
						An_OverNGStep:=1691;
					END_IF	
				END_IF				
		1691:
			    IF 	arrAxisCtrl[AxiseNo.AxisName.LeftYDUpDown].Cmd.arrbRealPoint[1] AND (arrAxisCtrl[AxiseNo.AxisName.RightYDUpDown].Cmd.arrbRealPoint[1] OR arrAxisCtrl[AxiseNo.AxisName.RightYDUpDown].Cmd.arrbRealPoint[15] ) AND
					    arrCyCtrl[arrCyNo.CylinderName.AnScrapbinCy].Status.ONState  AND arrCyCtrl[arrCyNo.CylinderName.CaScrapbinUDCy].Status.OFFState AND
                        arrCyCtrl[arrCyNo.CylinderName.PoleHotCutterCy].Status.OFFState   THEN
					An_OverNGStep:=1695;
				END_IF	
		
		    1695://				
					IF An_CarryingPos2 THEN//正极在叠片位
							An_OverNGStep:=1700;//
					ELSIF An_CarryingPos1  THEN//正极在取片位
							 An_OverNGStep:=1800;//
					ELSE
						  DTPosError[11]:=TRUE;//踢正极对齐度NG片 时，正极取片即不在取片位，也不在叠片位
					END_IF;
		
	

	        1800://	调用正极NG踢废		
                    DT_TON[2].IN:=FALSE;	
					CCD.Over.Start.iPhotoDo:=2;
					CCD.Over.Finish.OverhandResult:=0;
					Mach_Control.DT_b.OverhandResult:=0;
					Mach_Control.DT_b.CDD_OverStart:=TRUE;
					
			        Mach_Control.An_b.An_Quantited:=Mach_Control.An_b.An_Quantited-1;//正极已叠片数减一
                    An_Step2:=10; 
                    An_OverNGStep:=1810;

			1810://判断负极叠台搬运是否有片，有片的话放到纠偏台
			         DT_TON[2].IN:=TRUE;	
						IF arrCyCtrl[arrCyNo.ElectValveName.CaDTCarryingVacuum].Io.DIOnSwitch AND  Mach_Control.Ca_b.Ca_DPCarryingFalg  THEN//负极再取片位且叠台搬运有片,把当前片放到纠偏台
							An_OverNGStep:=1820;
						ELSE
							An_OverNGStep:=1850;	
						END_IF
	
			1820://纠偏台回初始位
				//纠偏平台X1移动至初始位
				IF NOT DP_SinStepe THEN
					IF arrAxisCtrl[AxiseNo.AxisName.CadeviationX1].Status.Homed  AND arrAxisCtrl[AxiseNo.AxisName.CadeviationX1].Status.NoMoving AND NOT  arrAxisCtrl[AxiseNo.AxisName.CadeviationX1].Status.Error THEN
						IF arrAxisCtrl[AxiseNo.AxisName.CadeviationX1].Cmd.arrbRealPoint[1] THEN
							arrAxisCtrl[AxiseNo.AxisName.CadeviationX1].Cmd.iGoSetPos:=0;
						ELSE
							arrAxisCtrl[AxiseNo.AxisName.CadeviationX1].Cmd.iGoSetPos:=1;
						END_IF					
					END_IF
					//纠偏平台X2移动至初始位
					IF arrAxisCtrl[AxiseNo.AxisName.CadeviationX2].Status.Homed  AND arrAxisCtrl[AxiseNo.AxisName.CadeviationX2].Status.NoMoving AND NOT  arrAxisCtrl[AxiseNo.AxisName.CadeviationX2].Status.Error THEN
						IF arrAxisCtrl[AxiseNo.AxisName.CadeviationX2].Cmd.arrbRealPoint[1] THEN
							arrAxisCtrl[AxiseNo.AxisName.CadeviationX2].Cmd.iGoSetPos:=0;
						ELSE
							arrAxisCtrl[AxiseNo.AxisName.CadeviationX2].Cmd.iGoSetPos:=1;
						END_IF					
					END_IF
					//纠偏平台X2移动至初始位
					IF arrAxisCtrl[AxiseNo.AxisName.CadeviationY].Status.Homed  AND arrAxisCtrl[AxiseNo.AxisName.CadeviationY].Status.NoMoving AND NOT  arrAxisCtrl[AxiseNo.AxisName.CadeviationY].Status.Error THEN
						IF arrAxisCtrl[AxiseNo.AxisName.CadeviationY].Cmd.arrbRealPoint[1] THEN
							arrAxisCtrl[AxiseNo.AxisName.CadeviationY].Cmd.iGoSetPos:=0;
						ELSE
							arrAxisCtrl[AxiseNo.AxisName.CadeviationY].Cmd.iGoSetPos:=1;
						END_IF					
					END_IF
					IF arrAxisCtrl[AxiseNo.AxisName.CadeviationX1].Cmd.arrbRealPoint[1] AND arrAxisCtrl[AxiseNo.AxisName.CadeviationX2].Cmd.arrbRealPoint[1] AND arrAxisCtrl[AxiseNo.AxisName.CadeviationY].Cmd.arrbRealPoint[1] THEN
						DT_SingeMode();//单步选择	
						An_OverNGStep:=1830;	
						DT_TON[4].IN:=FALSE;
					END_IF	
				END_IF
			1830://叠台搬运极片放回纠偏台
				IF NOT DP_SinStepe THEN
					IF arrAxisCtrl[AxiseNo.AxisName.CaDTCarryingLine].Cmd.arrbRealPoint[1]  AND NOT Mach_Control.Ca_b.Ca_deviationFalg THEN 
						IF arrAxisCtrl[AxiseNo.AxisName.CaDTCarryingUpDown].Cmd.arrbRealPoint[2] THEN
							arrAxisCtrl[AxiseNo.AxisName.CaDTCarryingUpDown].Cmd.iGoSetPos:=0;
					    ELSE
							arrAxisCtrl[AxiseNo.AxisName.CaDTCarryingUpDown].Cmd.iGoSetPos:=2;//负极d叠台搬运下降至取片位
					    END_IF
                   END_IF
				       IF arrAxisCtrl[AxiseNo.AxisName.CaDTCarryingUpDown].Cmd.arrbRealPoint[2] THEN
				           	/// 吸盘破真空    纠偏台开真空
							arrCyCtrl[arrCyNo.ElectValveName.CaDTCarryingVacuum].Cmd.bON:=TRUE;	//负极叠台搬运升降真空	真空
							arrCyCtrl[arrCyNo.ElectValveName.CaDTCarryingVacuum].Cmd.bOFF:=FALSE;	//负极叠台搬运升降真空破真空								
							arrCyCtrl[arrCyNo.ElectValveName.CadeviationVacuum].Cmd.bON:=TRUE;	//负极纠偏台真空			
							arrCyCtrl[arrCyNo.ElectValveName.CadeviationVacuum].Cmd.bOFF:=FALSE;	//负极纠偏台真空	   
							DT_SingeMode();//单步选择	
							An_OverNGStep:=1840;
							DT_TON[4].IN:=TRUE;
							Mach_Control.Ca_b.Ca_deviationFalg:=TRUE;//置位位纠偏平台有料标记
							Mach_Control.Ca_b.Ca_DPCarryingFalg:=FALSE;//负极搬运真空吸盘有料标记复位
	                    END_IF
				END_IF
			1840://叠台搬运极片上升至凸轮耦合初始高度
				IF NOT DP_SinStepe THEN
					IF arrAxisCtrl[AxiseNo.AxisName.CaDTCarryingUpDown].Cmd.arrbRealPoint[4] AND DT_TON[4].Q THEN
						arrAxisCtrl[AxiseNo.AxisName.CaDTCarryingUpDown].Cmd.iGoSetPos:=0;
						/// 吸盘破真空    纠偏台开真空
						Mach_Control.Ca_b.Ca_deviationFalg:=TRUE;//置位位纠偏平台有料标记
						Mach_Control.Ca_b.Ca_DPCarryingFalg:=FALSE;//负极搬运真空吸盘有料标记复位
						Par.stDT_date.Ca_MQ_Slice[8]:=Par.stDT_date.Ca_MQ_Slice[9];
						DT_SingeMode();//单步选择	
						An_OverNGStep:=1850;
						DT_TON[4].IN:=FALSE;
					ELSE
						arrAxisCtrl[AxiseNo.AxisName.CaDTCarryingUpDown].Cmd.iGoSetPos:=4;//负极搬运升降2上升至凸轮耦合初始高度
					END_IF			
				END_IF		   
		

			
	        1860://等待正极NG踢废完成		
  
				
					 IF 	An_Step2=6666 THEN
						    An_OverNGStep:=0;
							DP_Step0:=0;
                           // An_OverNGMark:=FALSE;	
					 END_IF
	  END_CASE
END_IF

 CASE An_OverNGStep OF  
	 
		1850://
                  
				   IF Mach_Control.DT_b.OverhandResult<>3 AND  DT_TON[2].Q THEN
					  Mach_Control.An_b.Error[22]:=TRUE;//正极叠台搬运升降真空报警，电芯上有片，请拿掉 
				   END_IF
			
				 IF 	 Mach_Control.DT_b.OverhandResult=3 THEN
					     DT_TON[2].IN:=FALSE;	
						An_OverNGStep:=1860;
				 END_IF
 
 
 
 
     1200: //正到负取正极NG对其度片,	正极搬运与叠片各轴在初始位,负极在叠片位
	             VirMain_TON.IN:=FALSE;   
				//正到负_正极送片搬运平移轴凸轮耦合
				fbAnCamInCarryingLine.ParCamIn.SlaveScaling:=1;
				fbAnCamInCarryingLine.bCamInExecute:=TRUE;	
		    	fbAnCamInCarryingUpDown.iTableSel:=3;      //20240528SJ
                fbAnCamInCarryingUpDown.bCamInExecute:=TRUE;
			//正到负_正极叠片平移轴凸轮耦合
				fbAnCamInDTCarryingLine.ParCamIn.SlaveScaling:=1;
				fbAnCamInDTCarryingLine.bCamInExecute:=TRUE;			
                fbAnCamInDTCarryingUpDown.iTableSel:=3;   //  //20240528SJ
                fbAnCamInDTCarryingUpDown.bCamInExecute:=TRUE;
			//正到负_正极搬运旋转轴凸轮耦合		
				fbAnCamInCarryingWhirling.ParCamIn.SlaveScaling:=1;
				fbAnCamInCarryingWhirling.bCamInExecute:=TRUE;						
			
			//正到负_负极送片搬运平移轴凸轮耦合
				fbCaCamInCarryingLine2.ParCamIn.SlaveScaling:=-1;
				fbCaCamInCarryingLine2.bCamInExecute:=TRUE;
			   fbCaCamInCarryingUpDown2.iTableSel:=3; //20240528SJ
               fbCaCamInCarryingUpDown2.bCamInExecute:=TRUE;
			//正到负_负极叠片搬运平移轴凸轮耦合
				fbCaCamInDTCarryingLine.ParCamIn.SlaveScaling:=-1;
				fbCaCamInDTCarryingLine.bCamInExecute:=TRUE;
			    fbCaCamInDTCarryingUpDown.iTableSel:=3;  //20240528SJ
                fbCaCamInDTCarryingUpDown.bCamInExecute:=TRUE;
			//正到负_ 缓存轴轮耦合
				fbCamInGMBuffer2.iTableSel:=1;
				 fbCamInGMBuffer2.bCamInExecute:=TRUE;
			//正到负_隔膜平移轴凸轮耦合
				fbCamInGMDanserMove.iTableSel:=1;
				fbCamInGMDanserMove.bCamInExecute:=TRUE;
			
			//正到负_放卷虚轴凸轮耦合
				 fbCamInVirGMDriver2.iTableSel :=1;
				 fbCamInVirGMDriver2.bCamInExecute:=TRUE;		
					
					//判断凸轮是否耦合完成
						IF  fbAnCamInCarryingLine.bInSync  AND  fbAnCamInDTCarryingLine.bInSync AND fbAnCamInCarryingWhirling.bInSync AND 
							 fbCaCamInCarryingLine2.bInSync AND fbCaCamInDTCarryingLine.bInSync AND
							 fbCamInGMBuffer2.bInSync AND fbCamInGMDanserMove.bInSync AND 
							 fbCamInVirGMDriver2.bInSync   AND
							 fbAnCamInCarryingUpDown.bInSync AND fbAnCamInDTCarryingUpDown.bInSync AND fbCaCamInCarryingUpDown2.bInSync AND fbCaCamInDTCarryingUpDown.bInSync AND  
                            Mach_Control.U.DT_iMode=1  THEN
							An_OverNGStep:=1210;//
						ELSIF   fbAnCamInCarryingLine.bError  OR  fbAnCamInDTCarryingLine.bError OR 
							 fbCaCamInCarryingLine2.bError OR fbCaCamInDTCarryingLine.bError OR
							 fbCamInGMBuffer2.bError OR fbCamInGMDanserMove.bError OR 
							  fbAnCamInCarryingUpDown.bError OR fbAnCamInDTCarryingUpDown.bError OR fbCaCamInCarryingUpDown2.bError OR fbCaCamInDTCarryingUpDown.bError OR  
							 fbCamInVirGMDriver2.bError THEN
								Mach_Control.DT_b.Error[19]:=TRUE;//凸轮耦合报警
								An_OverNGStep:=9991;										
						END_IF		
			1210://主轴启动
									arrAxisCtrl[AxiseNo.VirAxisName.VirMain].Cmd	.bDynamitcsParSel:=2;
									arrAxisPar[AxiseNo.VirAxisName.VirMain].fTagatTime:=VirMain_TagatTime;
									arrAxisCtrl[AxiseNo.VirAxisName.VirMain].Cmd	.fPositon_of_Abs:=360;
									arrAxisCtrl[AxiseNo.VirAxisName.VirMain].Cmd	.bMoveAbs:=TRUE;		
									
									IF  arrAxis[AxiseNo.VirAxisName.VirMain].Status.Moving AND arrAxisCtrl[AxiseNo.VirAxisName.VirMain].Status.fActPos>=10  THEN
										VirMain_TON.IN:=FALSE;
										arrAxisCtrl[AxiseNo.VirAxisName.VirMain].Cmd	.bMoveAbs:=FALSE;	
										An_OverNGStep:=1500;	
									ELSE
										IF NOT VirMain_TON.Q THEN
											VirMain_TON.IN:=TRUE;
										ELSE
											VirMain_TON.IN:=FALSE;
											Mach_Control.DT_b.Error[22]:=TRUE;//主轴启动超时报警
											An_OverNGStep:=10001;	
									END_IF	
				 	    END_IF		

           1300: //正到负取正极NG对其度片,正极搬运与叠片各轴在初始位,, 负极在取片位,  隔膜平移在负极位
		              VirMain_TON.IN:=FALSE;
						//正到负_正极送片搬运平移轴凸轮耦合
					fbAnCamInCarryingLine.ParCamIn.SlaveScaling:=1;
					fbAnCamInCarryingLine.bCamInExecute:=TRUE;					
					fbAnCamInCarryingUpDown.iTableSel:=3;      //20240528SJ
					fbAnCamInCarryingUpDown.bCamInExecute:=TRUE;
				//正到负_正极叠片平移轴凸轮耦合
					fbAnCamInDTCarryingLine.ParCamIn.SlaveScaling:=1;
					fbAnCamInDTCarryingLine.bCamInExecute:=TRUE;		
					fbAnCamInDTCarryingUpDown.iTableSel:=3;   //  //20240528SJ
					fbAnCamInDTCarryingUpDown.bCamInExecute:=TRUE;

			//正到负_正极搬运旋转轴凸轮耦合		
				fbAnCamInCarryingWhirling.ParCamIn.SlaveScaling:=1;
				fbAnCamInCarryingWhirling.bCamInExecute:=TRUE;							
								
					//判断凸轮是否耦合完成
						IF  fbAnCamInCarryingLine.bInSync AND fbAnCamInDTCarryingLine.bInSync AND  fbAnCamInCarryingWhirling.bInSync  AND 
                            fbAnCamInCarryingUpDown.bInSync AND  fbAnCamInDTCarryingUpDown.bInSync AND 
                            Mach_Control.U.DT_iMode=1 THEN
							An_OverNGStep:=1310;//
						ELSIF fbAnCamInCarryingLine.bError OR  fbAnCamInDTCarryingLine.bError  OR   fbAnCamInCarryingUpDown.bError OR   fbAnCamInDTCarryingUpDown.bError   THEN
								Mach_Control.DT_b.Error[19]:=TRUE;//凸轮耦合报警
								An_OverNGStep:=9992;										
						END_IF			   
		   
			1310://主轴启动
									arrAxisCtrl[AxiseNo.VirAxisName.VirMain].Cmd	.bDynamitcsParSel:=2;
									arrAxisPar[AxiseNo.VirAxisName.VirMain].fTagatTime:=VirMain_TagatTime;
									arrAxisCtrl[AxiseNo.VirAxisName.VirMain].Cmd	.fPositon_of_Abs:=360;
									arrAxisCtrl[AxiseNo.VirAxisName.VirMain].Cmd	.bMoveAbs:=TRUE;			
						
									IF  arrAxis[AxiseNo.VirAxisName.VirMain].Status.Moving AND arrAxisCtrl[AxiseNo.VirAxisName.VirMain].Status.fActPos>=10  THEN
										VirMain_TON.IN:=FALSE;
										arrAxisCtrl[AxiseNo.VirAxisName.VirMain].Cmd	.bMoveAbs:=FALSE;	
										An_OverNGStep:=1500;	
									ELSE
										IF NOT VirMain_TON.Q THEN
											VirMain_TON.IN:=TRUE;
										ELSE
											VirMain_TON.IN:=FALSE;
											Mach_Control.DT_b.Error[22]:=TRUE;//主轴启动超时报警
											An_OverNGStep:=10002;	
									END_IF	
				 	    END_IF							
										
	       1400: //正到负取正极NG对其度片,正极搬运与叠片各轴在初始位,, 负极在取片位,  隔膜平移在正极位	
			              VirMain_TON.IN:=FALSE;
						//正到负_正极送片搬运平移轴凸轮耦合
						fbAnCamInCarryingLine.ParCamIn.SlaveScaling:=1;
						fbAnCamInCarryingLine.bCamInExecute:=TRUE;				
						fbAnCamInCarryingUpDown.iTableSel:=3;      //20240528SJ
						fbAnCamInCarryingUpDown.bCamInExecute:=TRUE;

					//正到负_正极叠片平移轴凸轮耦合
						fbAnCamInDTCarryingLine.ParCamIn.SlaveScaling:=1;
						fbAnCamInDTCarryingLine.bCamInExecute:=TRUE;
					   fbAnCamInDTCarryingUpDown.iTableSel:=3;   //  //20240528SJ
                       fbAnCamInDTCarryingUpDown.bCamInExecute:=TRUE;
						
						
					//正到负_正极搬运旋转轴凸轮耦合		
						fbAnCamInCarryingWhirling.ParCamIn.SlaveScaling:=1;
						fbAnCamInCarryingWhirling.bCamInExecute:=TRUE;						
						
					//正到负_ 缓存轴轮耦合
						fbCamInGMBuffer2.iTableSel:=1;
						 fbCamInGMBuffer2.bCamInExecute:=TRUE;
						 
					//正到负_隔膜平移轴凸轮耦合
						fbCamInGMDanserMove.iTableSel:=1;
						fbCamInGMDanserMove.bCamInExecute:=TRUE;
						
					//正到负_放卷虚轴凸轮耦合
						 fbCamInVirGMDriver2.iTableSel :=1;
						 fbCamInVirGMDriver2.bCamInExecute:=TRUE;			   
						
					//判断凸轮是否耦合完成
						IF   fbAnCamInCarryingLine.bInSync  AND  fbAnCamInDTCarryingLine.bInSync AND   fbAnCamInCarryingWhirling.bInSync AND
							 fbCamInGMBuffer2.bInSync AND fbCamInGMDanserMove.bInSync AND 
							 fbAnCamInCarryingUpDown.bInSync AND fbAnCamInDTCarryingUpDown.bInSync AND 
							 fbCamInVirGMDriver2.bInSync  AND 
                            Mach_Control.U.DT_iMode=1  THEN
							An_OverNGStep:=1410;//
						ELSIF  fbAnCamInCarryingLine.bError  OR  fbAnCamInDTCarryingLine.bError OR 
							     fbCamInGMBuffer2.bError OR fbCamInGMDanserMove.bError OR 
								 fbAnCamInCarryingUpDown.bError OR  fbAnCamInDTCarryingUpDown.bError OR
							     fbCamInVirGMDriver2.bError THEN
										Mach_Control.DT_b.Error[19]:=TRUE;//凸轮耦合报警
										An_OverNGStep:=9993;										
						END_IF		
	
			1410://主轴启动
									arrAxisCtrl[AxiseNo.VirAxisName.VirMain].Cmd	.bDynamitcsParSel:=2;
									arrAxisPar[AxiseNo.VirAxisName.VirMain].fTagatTime:=VirMain_TagatTime;
									arrAxisCtrl[AxiseNo.VirAxisName.VirMain].Cmd	.fPositon_of_Abs:=360;
									arrAxisCtrl[AxiseNo.VirAxisName.VirMain].Cmd	.bMoveAbs:=TRUE;					
									IF  arrAxis[AxiseNo.VirAxisName.VirMain].Status.Moving AND arrAxisCtrl[AxiseNo.VirAxisName.VirMain].Status.fActPos>=10  THEN
										VirMain_TON.IN:=FALSE;
										arrAxisCtrl[AxiseNo.VirAxisName.VirMain].Cmd	.bMoveAbs:=FALSE;	
										An_OverNGStep:=1500;	
									ELSE
										IF NOT VirMain_TON.Q THEN
											VirMain_TON.IN:=TRUE;
										ELSE
											VirMain_TON.IN:=FALSE;
											Mach_Control.DT_b.Error[22]:=TRUE;//主轴启动超时报警
											An_OverNGStep:=10003;	
									END_IF	
				 	    END_IF							
   
			1500://
				(*IF 	arrAxisCtrl[AxiseNo.VirAxisName.VirMain].Status.fActPos>230 AND  arrAxisCtrl[AxiseNo.VirAxisName.VirMain].Status.fActPos<240 AND Mach_Control.Ca_b.Ca_DPCarryingFalg  THEN//198
					IF Mach_Control.DT_b.DT_CCD_TwoModel THEN
							CCD.CaRec.Finish.RectifyX1:=0;
							CCD.CaRec.Finish.RectifyX2:=0;
							CCD.CaRec.Finish.RectifyY:=0;		
							CCD.CaRec.Finish.RectifyResult:=0;//拍照结果清零									
							Mach_Control.Ca_b.Ca_CCDStart :=TRUE;//启动CCD拍照
							CCD.CaRec.Start.iPhotoDo:=2;//启动CCD第二次拍照									
					END_IF			
				END_IF	*)		
				
				IF arrAxis[AxiseNo.VirAxisName.VirMain].NcToPlc.SetPos=360 AND  arrAxis[AxiseNo.VirAxisName.VirMain].Status.NotMoving  THEN
					DP_Step1:=100;//解除耦合，主轴回零子程序			
					An_OverNGStep:=1510;	
				END_IF	
			1510://			
				IF NOT DP_SinStepe THEN
					IF DP_Step1=6666 AND arrAxis[AxiseNo.VirAxisName.VirMain].Status.NotMoving AND arrAxis[AxiseNo.VirAxisName.VirMain].NcToPlc.SetPos=0 AND NOT DT_AxiseCoupling  THEN
						DT_SingeMode();//单步选择
						An_OverNGStep:=1600;
					END_IF	
				END_IF	

		    1700://	/踢正极NG对齐度片回正极取片位,(正极轴不动 ) ,正极搬运叠片各轴在叠片位		
			         VirMain_TON.IN:=FALSE;
					//负到正_正极搬运平移轴凸轮耦合
					fbAnCamInCarryingLine.ParCamIn.SlaveScaling:=-1;
					fbAnCamInCarryingLine.bCamInExecute:=TRUE;
					fbAnCamInCarryingUpDown.iTableSel:=3;      //20240528SJ
                   fbAnCamInCarryingUpDown.bCamInExecute:=TRUE;
					
					//负到正_正极叠片平移轴凸轮耦合
					fbAnCamInDTCarryingLine.ParCamIn.SlaveScaling:=-1;
					fbAnCamInDTCarryingLine.bCamInExecute:=TRUE;	
					fbAnCamInDTCarryingUpDown.iTableSel:=3;   //  //20240528SJ
					fbAnCamInDTCarryingUpDown.bCamInExecute:=TRUE;

					//负到正_正极搬运旋转轴凸轮耦合
						fbAnCamInCarryingWhirling.ParCamIn.SlaveScaling:=-1;
						fbAnCamInCarryingWhirling.bCamInExecute:=TRUE;								
				
				IF fbAnCamInCarryingLine.bInSync  AND 
					fbAnCamInDTCarryingLine.bInSync  AND
					fbAnCamInCarryingWhirling.bInSync AND  
                    fbAnCamInCarryingUpDown.bInSync AND   fbAnCamInDTCarryingUpDown.bInSync AND  
                    Mach_Control.U.DT_iMode=1  THEN   
					DT_SingeMode();//单步选择		
					An_OverNGStep:=1710;
				ELSIF fbAnCamInCarryingLine.bError OR //  fbCaCamInCarryingUpDown2.bError or
					  fbAnCamInDTCarryingLine.bError  OR  fbAnCamInCarryingUpDown.bError OR    fbAnCamInDTCarryingUpDown.bError   THEN   
					Mach_Control.DT_b.Error[19]:=TRUE;//凸轮耦合报警
					An_OverNGStep:=9994;
				END_IF		

				1710://主轴启动
				      				
									arrAxisCtrl[AxiseNo.VirAxisName.VirMain].Cmd	.bDynamitcsParSel:=2;
									arrAxisPar[AxiseNo.VirAxisName.VirMain].fTagatTime:=VirMain_TagatTime;
									arrAxisCtrl[AxiseNo.VirAxisName.VirMain].Cmd	.fPositon_of_Abs:=360;
									arrAxisCtrl[AxiseNo.VirAxisName.VirMain].Cmd	.bMoveAbs:=TRUE;			
						IF  arrAxis[AxiseNo.VirAxisName.VirMain].Status.Moving AND arrAxisCtrl[AxiseNo.VirAxisName.VirMain].Status.fActPos>=10  THEN
							VirMain_TON.IN:=FALSE;
							arrAxisCtrl[AxiseNo.VirAxisName.VirMain].Cmd	.bMoveAbs:=FALSE;	
							An_OverNGStep:=1720;	
						ELSE
								IF NOT VirMain_TON.Q THEN
									VirMain_TON.IN:=TRUE;
								ELSE
									VirMain_TON.IN:=FALSE;
									Mach_Control.DT_b.Error[22]:=TRUE;//主轴启动超时报警
									An_OverNGStep:=10004;	
							END_IF	
					   END_IF				

			1720://
				IF arrAxis[AxiseNo.VirAxisName.VirMain].NcToPlc.SetPos=360 AND  arrAxis[AxiseNo.VirAxisName.VirMain].Status.NotMoving  THEN
					DP_Step1:=100;//解除耦合，主轴回零子程序			
					An_OverNGStep:=1730;	
				END_IF	
	
				
			1730://			
				IF NOT DP_SinStepe THEN
					IF DP_Step1=6666 AND arrAxis[AxiseNo.VirAxisName.VirMain].Status.NotMoving AND arrAxis[AxiseNo.VirAxisName.VirMain].NcToPlc.SetPos=0 AND NOT DT_AxiseCoupling  THEN
						DT_SingeMode();//单步选择
						An_OverNGStep:=1800;
					END_IF	
				END_IF	
									
 END_CASE
END_ACTION

ACTION An_Rectifydev:
rAnCCD_Ton(IN:= , PT:=T#1.5S , Q=> , ET=> );//正极CCD拍照超时报警
IF (NOT Mach_Control.An_b.An_deviationFalg AND Mach_Control.U.DT_iMode=1) AND NOT Mach_Control.An_b.Demarcateing   THEN
//IF NOT Mach_Control.An_b.An_deviationFalg THEN
	Mach_Control.An_b.RectifydevDone:=FALSE;
	An_CCD_Done:=FALSE;
	CCD.AnRec.Finish.RectifyX1:=0;
	CCD.AnRec.Finish.RectifyX2:=0;
	CCD.AnRec.Finish.RectifyY:=0;
END_IF

rAnCCD_Ton1(IN:=Mach_Control.An_b.An_CCDStart , PT:=T#0.1S , Q=> , ET=> );//正极CCD拍照启动复位
IF rAnCCD_Ton1.Q THEN
	Mach_Control.An_b.An_CCDStart :=FALSE;
END_IF


An_CQ_ton(IN:=arrCyCtrl[arrCyNo.ElectValveName.AndeviationIonizedWind].Io.DOStatus1 , PT:=T#0.3S , Q=> , ET=>);
IF An_CQ_ton.Q THEN
	Mach_Control.An_b.An_Rectifydev_CQ:=FALSE;
	arrCyCtrl[arrCyNo.ElectValveName.AndeviationIonizedWind].Cmd.bON:=FALSE;//正极纠偏平台除尘
	arrCyCtrl[arrCyNo.ElectValveName.AndeviationIonizedWind].Cmd.bOFF:=TRUE;//正极纠偏平台除尘
END_IF



IF rAnUse[2].Q THEN
	CCD.AnRec.Finish.RectifyResult:=0;
	CCD.AnRec.Finish.RectifyX1:=0;
	CCD.AnRec.Finish.RectifyX2:=0;
	CCD.AnRec.Finish.RectifyY:=0;												
END_IF



IF Mach_Control.U.DT_iMode=1 THEN//在自动状态下
//判断负极是否允许取纠偏
IF (Mach_Control.An_b.An_deviationFalg AND (An_CCD_Done OR Mach_Control.An_b.RectifydevDone)) (*AND CCD.AnRec.Finish.RectifyResult=1 AND Mach_Control.An_b.RectifydevDone)*) OR
	 (Mach_Control.An_b.An_deviationFalg AND CCD.AnRec.Finish.RectifyResult<>1 AND arrAxisCtrl[AxiseNo.AxisName.AndeviationX1].Cmd.arrbRealPoint[1] AND 	arrAxisCtrl[AxiseNo.AxisName.AndeviationX2].Cmd.arrbRealPoint[1]  AND 	arrAxisCtrl[AxiseNo.AxisName.AndeviationY].Cmd.arrbRealPoint[1] )OR
	(Mach_Control.U.CCD_ChosesHMI  OR Mach_Control.U.EmptyRunMode)	 THEN
	Mach_Control.An_b.An_deviationDPOK:=TRUE;//取正极 偏平台极片允许
ELSE
	Mach_Control.An_b.An_deviationDPOK:=FALSE;
END_IF 	

	CASE An_StandbyStep0 OF
			0://判断正极纠偏平台是否有极片
				IF Mach_Control.An_b.An_deviationFalg AND NOT Mach_Control.U.EmptyRunMode  THEN
						IF NOT An_CCD_Done THEN
							CCD.AnRec.Finish.RectifyResult:=0;
							CCD.AnRec.Finish.RectifyX1:=0;
							CCD.AnRec.Finish.RectifyX2:=0;
							CCD.AnRec.Finish.RectifyY:=0;
							iMD11:=1;
							An_StandbyStep0:=10;
						END_IF
				ELSE
						iMD11:=2;
						An_RecdevPla_Step0:=0;
						Mach_Control.An_b.RectifydevStart :=FALSE;
						An_StandbyStep0:=10;
				END_IF
			10://正极纠偏平台回初始位
			IF  NOT Mach_Control.U.EmptyRunMode THEN
					Mach_Control.An_b.RectifydevStart :=FALSE;//复位纠偏启动
					Mach_Control.An_b.RectifydevDone:=FALSE;//复位纠偏完成
					IF Mach_Control.An_b.CarryingSafepos[4] THEN
							//纠偏平台X1移动至初始位
							IF arrAxisCtrl[AxiseNo.AxisName.AndeviationX1].Status.Homed  AND arrAxisCtrl[AxiseNo.AxisName.AndeviationX1].Status.NoMoving AND NOT  arrAxisCtrl[AxiseNo.AxisName.AndeviationX1].Status.Error THEN
								IF arrAxisCtrl[AxiseNo.AxisName.AndeviationX1].Cmd.arrbRealPoint[1] THEN
									arrAxisCtrl[AxiseNo.AxisName.AndeviationX1].Cmd.iGoSetPos:=0;
								ELSE
									arrAxisCtrl[AxiseNo.AxisName.AndeviationX1].Cmd.iGoSetPos:=1;
								END_IF					
							END_IF
							//纠偏平台X2移动至初始位
							IF arrAxisCtrl[AxiseNo.AxisName.AndeviationX2].Status.Homed  AND arrAxisCtrl[AxiseNo.AxisName.AndeviationX2].Status.NoMoving AND NOT  arrAxisCtrl[AxiseNo.AxisName.AndeviationX2].Status.Error THEN
								IF arrAxisCtrl[AxiseNo.AxisName.AndeviationX2].Cmd.arrbRealPoint[1] THEN
									arrAxisCtrl[AxiseNo.AxisName.AndeviationX2].Cmd.iGoSetPos:=0;
								ELSE
									arrAxisCtrl[AxiseNo.AxisName.AndeviationX2].Cmd.iGoSetPos:=1;
								END_IF					
							END_IF
							//纠偏平台X2移动至初始位
							IF arrAxisCtrl[AxiseNo.AxisName.AndeviationY].Status.Homed  AND arrAxisCtrl[AxiseNo.AxisName.AndeviationY].Status.NoMoving AND NOT  arrAxisCtrl[AxiseNo.AxisName.AndeviationY].Status.Error THEN
								IF arrAxisCtrl[AxiseNo.AxisName.AndeviationY].Cmd.arrbRealPoint[1] THEN
									arrAxisCtrl[AxiseNo.AxisName.AndeviationY].Cmd.iGoSetPos:=0;
								ELSE
									arrAxisCtrl[AxiseNo.AxisName.AndeviationY].Cmd.iGoSetPos:=1;
								END_IF					
							END_IF	
							IF 	 arrAxisCtrl[AxiseNo.AxisName.AndeviationX1].Cmd.arrbRealPoint[1] AND 	arrAxisCtrl[AxiseNo.AxisName.AndeviationX2].Cmd.arrbRealPoint[1]  AND 	arrAxisCtrl[AxiseNo.AxisName.AndeviationY].Cmd.arrbRealPoint[1] THEN
									IF  iMD11=1 THEN
											 An_StandbyStep0:=101;
											 rAnCCD_Ton.IN:=FALSE;
									 ELSIF  iMD11=2 THEN
											An_StandbyStep0:=0;
									 END_IF  			
							END_IF						
					END_IF
	END_IF
			101:
					CCD.AnRec.Finish.RectifyResult:=0;
					Mach_Control.An_b.An_CCDStart :=TRUE;//启动CCD拍照						
					CCD.AnRec.Start.iPhotoDo:=1;//第一次拍照	
					CCD.AnRec.Start.stPoleNo:=Par.stDT_date.An_MQ_Slice[1].stPoleNo;	
					An_StandbyStep0:=110;	
			110:
					IF NOT rAnCCD_Ton.Q THEN						
						rAnCCD_Ton.IN:=TRUE;
						IF Mach_Control.An_b.An_deviationCCDDone OR Mach_Control.U.CCD_ChosesHMI THEN
							rAnCCD_Ton.IN:=FALSE;
							An_CCD_Done:=TRUE;
							An_StandbyStep0:=111;
						END_IF
					ELSE
							rAnCCD_Ton.IN:=FALSE;
							Mach_Control.An_b.Error[7]:=TRUE;//正极CCD第一次拍照超时
							An_StandbyStep0:=9999;
					END_IF
			
			111://启动拍照			
					Mach_Control.An_b.An_CCDStart :=FALSE;//启动CCD拍照						
					rAnCCD_Ton.IN:=FALSE;
					An_StandbyStep0:=0;					

	END_CASE
ELSE
//正极纠偏平台CCD标定自动
IF Mach_Control.An_b.DemarcateStart THEN
	CCD.AnRec.Start.iPhotoDo:=1;//第一次拍照	
END_IF
An_Demarcate(
	Step0:=An_Demarcate_Step0,
	AxisX1_NO:=AxiseNo.AxisName.AndeviationX1 , //正极纠偏X1轴号
	AxisX2_NO:=AxiseNo.AxisName.AndeviationX2 , //正极纠偏X2轴号
	AxisY_NO:=AxiseNo.AxisName.AndeviationY , //正极纠偏Y轴号
	DemarcateStart:=Mach_Control.An_b.DemarcateStart , //纠偏平台CCD标定启动
	CCDStart:=Mach_Control.An_b.An_CCDStart , //CCD拍照启动
	CCDNo:=CCD.AnRec.iDemCount,//CCD拍照次数
	DemarcateResult:=CCD.AnRec.iDemarcatResult,//标定结果
	DemarcateDone:=Mach_Control.An_b.DemarcateDone ,//CCD标定完成
	Demarcateing:=Mach_Control.An_b.Demarcateing,	//CCD标定中
	Error :=Mach_Control.An_b.Error[8]  );//CCD标定NG
END_IF
//正极纠偏自动
rAn_RecdevPlaR_TRIG(CLK:=Mach_Control.An_b.An_deviationFalg AND (CCD.AnRec.Finish.RectifyResult=1 OR CCD.AnRec.Finish.RectifyResult=2 ) AND NOT Mach_Control.U.CCD_ChosesHMI AND NOT Mach_Control.An_b.RectifydevDone AND 
										 		(CCD.AnRec.Finish.RectifyX1<>0 OR CCD.AnRec.Finish.RectifyX2<>0 OR CCD.AnRec.Finish.RectifyY<>0) AND CCD.AnRec.Start.iPhotoDo=1  , Q=> );//AND NOT Mach_Control.An_b.An_VacuumErrorNG
IF rAn_RecdevPlaR_TRIG.Q  THEN//AND NOT Blueflaging
	Mach_Control.An_b.RectifydevStart:=TRUE;
END_IF

//纠偏结果限定
IF (CCD.AnRec.Finish.RectifyX1>=15 OR CCD.AnRec.Finish.RectifyX2>=15 OR CCD.AnRec.Finish.RectifyY>=10 OR
	CCD.AnRec.Finish.RectifyX1<=-15 OR CCD.AnRec.Finish.RectifyX2<=-15 OR CCD.AnRec.Finish.RectifyY<=-10) AND NOT Mach_Control.An_b.Demarcateing THEN
	CCD.AnRec.Finish.RectifyX1:=0;
	CCD.AnRec.Finish.RectifyX2:=0;
	CCD.AnRec.Finish.RectifyY:=0;
END_IF


CCD.AnRec.Finish.Offset_X:=fCaOffsetMean_X;
CCD.AnRec.Finish.Offset_Y:=fCaOffsetMean_Y;

An_RecdevPla(
	Step0:=An_RecdevPla_Step0,
	RecdevStart:=Mach_Control.An_b.RectifydevStart , //正极纠偏平台纠偏启动
	RecdevDone:=Mach_Control.An_b.RectifydevDone , //正极纠偏平台纠偏完成
	RecdevAgree:=Mach_Control.An_b.CarryingSafepos[4] , //正极纠偏平台纠偏允许
	AxisX1_NO:=AxiseNo.AxisName.AndeviationX1  , //正极纠偏平台X1轴号
	AxisX2_NO:=AxiseNo.AxisName.AndeviationX2 , //正极纠偏平台X2轴号
	AxisY_NO:=AxiseNo.AxisName.AndeviationY  , //正极纠偏平台Y轴号
	CCD_X1:=CCD.AnRec.Finish.RectifyX1 ,//正极纠偏平台X1纠偏量
	CCD_X2:=CCD.AnRec.Finish.RectifyX2 , //正极纠偏平台X2纠偏量
	CCD_Y:=CCD.AnRec.Finish.RectifyY );//正极纠偏平台Y纠偏量
	
//纠偏平台重复精度测试
AN_RectifyTry_fb(
	Execute:=Mach_Control.An_b.RectifyTryStart AND Mach_Control.U.DT_iMode=3 , //纠偏平台重复精度测试启动 
	AxisNO_X:=AxiseNo.AxisName.AndeviationX1 , 
	AxisNO_Y:= AxiseNo.AxisName.AndeviationX2, 
	AxisNO_R:=AxiseNo.AxisName.AndeviationY , 
	Demarcate_X:=Par.stDT_date.An_Demarcate_X , //纠偏平台重复精度测试X纠偏量
	Demarcate_Y:=Par.stDT_date.An_Demarcate_Y , //纠偏平台重复精度测试Y纠偏量
	Demarcate_R:=Par.stDT_date.An_Demarcate_R ,  //纠偏平台重复精度测试R纠偏量
	CCDNo:=Par.stDT_date.An_CCDNo, //纠偏平台重复精度测试次数
	CCDStart:= Mach_Control.An_b.An_CCDStart );
	
//吸盘重复精度测试		
An_SuckerTest_fb(
	Execute:=Mach_Control.An_b.SuckerTestStart AND Mach_Control.U.DT_iMode=3 , //吸盘重复精度测试启动 , 
	AxisNO_1:= AxiseNo.AxisName.AnDTCarryingUpDown, 
	AxisNO_2:=AxiseNo.AxisName.AnDTCarryingLine , 
	AxisNO_X:= AxiseNo.AxisName.AndeviationX1 , 
	AxisNO_Y:= AxiseNo.AxisName.AndeviationX2, 
	AxisNO_R:= AxiseNo.AxisName.AndeviationY , 
	DTCarryingVacuum:=arrCyNo.ElectValveName.AnDTCarryingVacuum , 
	deviationVacuum:= arrCyNo.ElectValveName.AndeviationVacuum, 
	deviationVacuumBark:=arrCyNo.ElectValveName.AndeviationVacuumBark, 
	CCDCount:= Par.stDT_date.An_CCDCount, //吸盘重复精度测试次数
	CCDStart:=Mach_Control.An_b.An_CCDStart,	
	CCD_X1:=CCD.AnRec.Finish.RectifyX1 ,//正极纠偏平台X1纠偏量
	CCD_X2:=CCD.AnRec.Finish.RectifyX2 , //正极纠偏平台X2纠偏量
	CCD_Y:=CCD.AnRec.Finish.RectifyY,//正极纠偏平台Y纠偏量
    DTiMode:= Mach_Control.U.DT_iMode  );
	
	//正极通讯监控
rtAn_CCDTest1(CLK:=Mach_Control.An_b.bAnCCD_TestDo , Q=> );
IF rtAn_CCDTest1.Q THEN
	bAn_CCDTest1:=FALSE;
	bAn_CCDTest2:=FALSE;
END_IF
IF Mach_Control.An_b.bAnCCD_TestDo THEN
	rtAn_CCDTest2(CLK:=Mach_Control.An_b.An_CCDStart , Q=> );
	rtAn_CCDTest3(CLK:=CCD.AnRec.Finish.RectifyResult<>0 , Q=> );
	rtAn_CCDTest4(CLK:=Mach_Control.An_b.An_deviationCCDDone , Q=> );
	IF rtAn_CCDTest2.Q THEN
		bAn_CCDTest1:=TRUE;
		bAn_CCDTest2:=TRUE;
		CCD.AnRec.Finish.RectifyResult:=0;
	END_IF
	IF rtAn_CCDTest3.Q THEN
		bAn_CCDTest1:=FALSE;
	END_IF	
	IF rtAn_CCDTest4.Q THEN
		bAn_CCDTest2:=FALSE;
	END_IF
	tonAn_CCDTest1(IN:=bAn_CCDTest1 , PT:=T#999MS , Q=> , ET=> );
	tonAn_CCDTest2(IN:=bAn_CCDTest2 , PT:=T#999MS , Q=> , ET=> );
	IF bAn_CCDTest1 THEN
		Mach_Control.An_b.iAnCCD_RectifyCT:= TIME_TO_INT(tonAn_CCDTest1.ET);
	END_IF
	IF bAn_CCDTest2 THEN
		Mach_Control.An_b.iAnCCD_PhotoCT:= TIME_TO_INT(tonAn_CCDTest2.ET);
	END_IF
	IF tonAn_CCDTest1.Q THEN
		Mach_Control.An_b.bAnCCD_TestDo:=FALSE;
	END_IF
END_IF
	
//正极白班NG计数
IF HMI_Hour>=8 AND HMI_Hour<20 AND An_Step2>50 AND An_Step2<70 THEN
  IF CCD.AnRec.Finish.NG_Code = 1 THEN
   CCD.AnRec.DayNgclassification.X1_NG :=CCD.AnRec.DayNgclassification.X1_NG+1 ;
   CCD.AnRec.Finish.NG_Code := 0 ;
  ELSIF CCD.AnRec.Finish.NG_Code = 2 THEN
   CCD.AnRec.DayNgclassification.X2_NG := CCD.AnRec.DayNgclassification.X2_NG+1 ;  
   CCD.AnRec.Finish.NG_Code := 0 ;
  ELSIF CCD.AnRec.Finish.NG_Code = 3 THEN
   CCD.AnRec.DayNgclassification.Y_NG := CCD.AnRec.DayNgclassification.Y_NG+1 ;  
   CCD.AnRec.Finish.NG_Code := 0 ;
  ELSIF CCD.AnRec.Finish.NG_Code = 4 THEN
   CCD.AnRec.DayNgclassification.R_NG := CCD.AnRec.DayNgclassification.R_NG+1 ;   
   CCD.AnRec.Finish.NG_Code := 0 ; 
  ELSIF CCD.AnRec.Finish.NG_Code = 5 THEN 
   CCD.AnRec.DayNgclassification.other_NG :=  CCD.AnRec.DayNgclassification.other_NG+1;
   CCD.AnRec.Finish.NG_Code := 0 ;
  END_IF	
END_IF  

DayClear1(CLK:=(HMI_Hour=8 AND HMI_Minute=0 AND HMI_Second=0 ) , Q=> );
NightClear1(CLK:=(HMI_Hour=20 AND HMI_Minute=0 AND HMI_Second=0) , Q=> );

//正极白班N清零
IF DayClear1.Q  THEN
  Par.stDT_date.An_Rectifydev_DayNG:=0;
END_IF 

IF CCD.AnRec.DayNgclassification.NgClear[1] OR DayClear1.Q  THEN
   CCD.AnRec.DayNgclassification.X1_NG :=0 ;
END_IF

IF CCD.AnRec.DayNgclassification.NgClear[2] OR DayClear1.Q  THEN
   CCD.AnRec.DayNgclassification.X2_NG :=0 ;
END_IF

IF CCD.AnRec.DayNgclassification.NgClear[3] OR DayClear1.Q  THEN
   CCD.AnRec.DayNgclassification.Y_NG :=0 ;
END_IF

IF CCD.AnRec.DayNgclassification.NgClear[4] OR DayClear1.Q  THEN
   CCD.AnRec.DayNgclassification.R_NG :=0 ;
END_IF	

IF CCD.AnRec.DayNgclassification.NgClear[5] OR DayClear1.Q  THEN
   CCD.AnRec.DayNgclassification.other_NG :=0 ;
END_IF	
	
//正极晚班NG计数
IF ((HMI_Hour>=0 AND HMI_Hour<8) OR  (HMI_Hour>=20 AND HMI_Hour<=23)) AND An_Step2>50 AND An_Step2<70  THEN
  IF CCD.AnRec.Finish.NG_Code = 1 THEN
   CCD.AnRec.NightNgclassification.X1_NG :=CCD.AnRec.NightNgclassification.X1_NG+1 ;
   CCD.AnRec.Finish.NG_Code := 0 ;
  ELSIF CCD.AnRec.Finish.NG_Code = 2 THEN
   CCD.AnRec.NightNgclassification.X2_NG := CCD.AnRec.NightNgclassification.X2_NG+1 ;  
   CCD.AnRec.Finish.NG_Code := 0 ;
  ELSIF CCD.AnRec.Finish.NG_Code = 3 THEN
   CCD.AnRec.NightNgclassification.Y_NG := CCD.AnRec.NightNgclassification.Y_NG+1 ;  
   CCD.AnRec.Finish.NG_Code := 0 ;
  ELSIF CCD.AnRec.Finish.NG_Code = 4 THEN
   CCD.AnRec.NightNgclassification.R_NG := CCD.AnRec.NightNgclassification.R_NG+1 ;   
   CCD.AnRec.Finish.NG_Code := 0 ; 
  ELSIF CCD.AnRec.Finish.NG_Code = 5 THEN 
   CCD.AnRec.NightNgclassification.other_NG :=  CCD.AnRec.NightNgclassification.other_NG+1;
   CCD.AnRec.Finish.NG_Code := 0 ;
  END_IF	
END_IF  

//正极晚班NG清零
IF  NightClear1.Q  THEN
   Par.stDT_date.An_Rectifydev_NightNG:=0;
END_IF

IF CCD.AnRec.NightNgclassification.NgClear[1] OR NightClear1.Q  THEN
   CCD.AnRec.NightNgclassification.X1_NG :=0 ;
END_IF

IF CCD.AnRec.NightNgclassification.NgClear[2] OR NightClear1.Q  THEN
   CCD.AnRec.NightNgclassification.X2_NG :=0 ;
END_IF

IF CCD.AnRec.NightNgclassification.NgClear[3] OR NightClear1.Q  THEN
   CCD.AnRec.NightNgclassification.Y_NG :=0 ;
END_IF

IF CCD.AnRec.NightNgclassification.NgClear[4] OR NightClear1.Q  THEN
   CCD.AnRec.NightNgclassification.R_NG :=0 ;
END_IF	

IF CCD.AnRec.NightNgclassification.NgClear[5] OR NightClear1.Q  THEN
   CCD.AnRec.NightNgclassification.other_NG :=0 ;
END_IF
END_ACTION

ACTION An_StandbyMain:
An_TON[1](PT:=T#0.5S);//正极拍照结果超时报警
An_TON[2](PT:=T#5S);//叠台主轴启动超时报警延时
An_TON[3](PT:=T#0.5S);
An_TON[5](PT:=T#10MS);
An_TON[6](PT:=T#0.2S);
An_TON[7](PT:=T#0.3S);
An_TON[8](PT:=T#0.3S);
An_TON[9](PT:=T#0.1S);
An_TON[10](PT:=T#2.5S);
An_TON[11](PT:=T#2.5S);
//An_StandbyStep1



